(* IEC 61131-3 sources: SRCI/RobotLibrary/Library/POUs/General/MC_RobotTask (part 4) *)

         // timeout exceeded ?
         IF (CheckTimeout(_rTimer) = RobotLibraryConstants.OK)
         THEN
           ErrorID     := RobotLibraryErrorIdEnum.ERR_TIMEOUT_CMD;
           ErrorAddTxt := CONCAT(_stepName, DINT_TO_STRING(_rStep));
         END_IF
       END_IF

       // Wait Tooldata read
    2: IF (( NOT _readToolData.Busy  ) AND
           ( NOT _readToolData.Error ) AND
           (     _readToolData.Done  ))
       THEN
         // reset execution
        _readToolData.Execute := FALSE;
         // set available bit
        _toolData[_rSyncIdx].Available := TRUE;
         ToolData[_rSyncIdx].Available := TRUE;
         // Copy data
        _toolData[_rSyncIdx].Data := _readToolData.OutCmd.ToolData;

         // Check tool data is equal ?
         IF ( NOT IsToolDataEqual( Data1 := _toolData[_rSyncIdx].Data, Data2 := ToolData[_rSyncIdx].Data, IgnoreTimestamp := TRUE))
         THEN
           // Reset plc in sync flag
           AxesGroup.State.SyncStatePlc.InSync.Tool := FALSE;
           // Set data changed flag
           AxesGroup.State.DataChanged.Tool[_rSyncIdx] := TRUE;
           // inc count of unsynchronised plc tools
           AxesGroup.State.SyncStatePlc.UnSyncNo.Tool := AxesGroup.State.SyncStatePlc.UnSyncNo.Tool + 1;

           // Create log entry
           CreateLogMessagePara1 ( Timestamp   := SystemTime,
                                   MessageType := MessageType.CMD,
                                   Severity    := Severity.DEBUG,
                                   MessageCode := 0,
                                   MessageText := 'SyncToolData: Detected a difference in Tool[{1}] between PLC and RC',
                                   Para1       :=  DINT_TO_STRING(_rSyncIdx));

           // Check synchronisation is enabled ?
           IF ( NOT AxesGroup.State.DataEnableSync.EnableSyncTool ) AND (InfoID = RobotLibraryInfoIdEnum.NO_INFO )
           THEN
             InfoID := RobotLibraryInfoIdEnum.INFO_SYNC_TOOL_DATA_DISABLED;
  				 END_IF

           // Check user interaction needed ?
           IF ( AxesGroup.Parameter.PLC.Parameter.SyncUserInteraction.Tool ) AND ( WarningID = RobotLibraryWarningIdEnum.NO_WARNING )
           THEN
             WarningID := RobotLibraryWarningIdEnum.WARN_TOOL_NUMBER_SYNC_ERROR;
  				 END_IF
  			 END_IF

         // Check all tools read ?
         IF ( _rSyncIdx < AxesGroup.State.UnifiedToolIndex )
         THEN
           // set timeout
           SetTimeout(PT := _rTimeout, rTimer := _rTimer);
           // inc tool index
          _rSyncIdx := _rSyncIdx + 1;
           // dec step counter
          _rStep := _rStep - 1;
         ELSE
           // set timeout
           SetTimeout(PT := _rTimeout, rTimer := _rTimer);
           // inc step counter
          _rStep := _rStep + 1;
         END_IF
       ELSE
         // check error ?
         IF (_readToolData.Error)
         THEN
           // Set warning
           WarningID := RobotLibraryWarningIdEnum.WARN_TOOL_SYNC_FAILED_BY_ERROR_OF_READ_OR_WRITE_CMD;
           // reset available bit
           ToolData[_rSyncIdx].Available := FALSE;
          _toolData[_rSyncIdx].Available := FALSE;
         END_IF

         // timeout exceeded ?
         IF (CheckTimeout(_rTimer) = RobotLibraryConstants.OK)
         THEN
           ErrorID     := RobotLibraryErrorIdEnum.ERR_TIMEOUT_CMD;
           ErrorAddTxt := CONCAT(_stepName, DINT_TO_STRING(_rStep));
         END_IF
       END_IF

       // Check synchronisation state ?
    3: IF (( AxesGroup.State.SyncStatePlc.UnSyncNo.Tool                                            = 0                           ) OR
           ( AxesGroup.Parameter.Plc.Parameter.SynchronizationModes.Tool[SyncTime.DURING_START_UP] = SyncMode.NO_SYNCHRONIZATION ))
       THEN
         // Update bit for data in sync
         AxesGroup.State.SyncStatePlc.InSync.Tool := (AxesGroup.State.SyncStatePlc.UnSyncNo.Tool = 0);
         // set timeout
         SetTimeout(PT := _rTimeout, rTimer := _rTimer);
         // inc step counter
        _rStep := 10; // -> jump to after startup

         // Create log entry
         CreateLogMessagePara1 ( Timestamp   := SystemTime,
                                 MessageType := MessageType.CMD,
                                 Severity    := Severity.DEBUG,
                                 MessageCode := 0,
                                 MessageText := 'SyncToolData: Synchronization Startup Phase done',
                                 Para1       :=  '' );
       ELSE
         // Check user interaction needed ?
         IF ( NOT AxesGroup.Parameter.PLC.Parameter.SyncUserInteraction.Tool )
         THEN
           CASE AxesGroup.Parameter.Plc.Parameter.SynchronizationModes.Tool[SyncTime.DURING_START_UP] OF

             SyncMode.SERVER_TO_CLIENT :

               // Overwrite PLC data with RC data
               ToolData := _toolData;
               // Reset data changed flags
               AxesGroup.State.DataChanged.Tool := _dataChangedNone.Tool;
               // Reset Synchronizing flag
               AxesGroup.State.Synchronizing.Tool := FALSE;
               // Set plc in sync flag
               AxesGroup.State.SyncStatePlc.InSync.Tool := TRUE;
               // Reset count of unsynchronised plc tools
               AxesGroup.State.SyncStatePlc.UnSyncNo.Tool := 0;
               // set timeout
               SetTimeout(PT := _rTimeout, rTimer := _rTimer);
               // inc step counter
              _rStep := 10; // -> jump to after startup

              // Create log entry
              CreateLogMessagePara3 ( Timestamp   := SystemTime,
                                      MessageType := MessageType.CMD,
                                      Severity    := Severity.DEBUG,
                                      MessageCode := 0,
                                      MessageText := 'SyncToolData: Synchronization of Tools triggered by StartUp-Compare, SyncMode = {2}, SyncTime = {3}, SyncDirection = RC -> PLC',
                                      Para1       :=  DINT_TO_STRING(_rSyncIdx),
                                      Para2       :=  SYNC_MODE_TO_STRING(AxesGroup.Parameter.Plc.Parameter.SynchronizationModes.Tool[SyncTime.DURING_START_UP]),
                                      Para3       :=  SYNC_TIME_TO_STRING(SyncTime.DURING_START_UP));
              // Create log entry
              CreateLogMessagePara1 ( Timestamp   := SystemTime,
                                      MessageType := MessageType.CMD,
                                      Severity    := Severity.DEBUG,
                                      MessageCode := 0,
                                      MessageText := 'SyncToolData: Applied the initial read tool data from RC',
                                      Para1       :=  '' );

  				   SyncMode.CLIENT_TO_SERVER : ;

               // Check conflicts to solve ?
               FOR _rSyncIdx := 0 TO AxesGroup.State.UnifiedToolIndex
               DO
                 IF ( AxesGroup.State.DataChanged.Tool[_rSyncIdx] )
                 THEN
                  _found := TRUE;
                   EXIT;
  		  			   END_IF
               END_FOR

               IF ( _found )
               THEN
                 // Reset plc in sync flag
                 AxesGroup.State.SyncStatePlc.InSync.Tool := FALSE;
                 // Set Synchronizing flag
                 AxesGroup.State.Synchronizing.Tool := TRUE;
                 // set timeout
                 SetTimeout(PT := _rTimeout, rTimer := _rTimer);
                 // inc step counter
                _rStep := _rStep +1; // -> write PLC data to RC
                 // Create log entry
                 CreateLogMessagePara3 ( Timestamp   := SystemTime,
                                         MessageType := MessageType.CMD,
                                         Severity    := Severity.DEBUG,
                                         MessageCode := 0,
                                         MessageText := 'SyncToolData: Synchronization of Tool[{1}] triggered by StartUp-Compare, SyncMode = {2}, SyncTime = {3}, SyncDirection = PLC -> RC',
                                         Para1       :=  DINT_TO_STRING(_rSyncIdx),
                                         Para2       :=  SYNC_MODE_TO_STRING(AxesGroup.Parameter.Plc.Parameter.SynchronizationModes.Tool[SyncTime.DURING_START_UP]),
                                         Para3       :=  SYNC_TIME_TO_STRING(SyncTime.DURING_START_UP));
               ELSE
                 // Reset data changed flags
                 AxesGroup.State.DataChanged.Tool := _dataChangedNone.Tool;
                 // Reset Synchronizing flag
                 AxesGroup.State.Synchronizing.Tool := FALSE;
                 // Set plc in sync flag
                 AxesGroup.State.SyncStatePlc.InSync.Tool := TRUE;
                 // Reset count of unsynchronised tools
                 AxesGroup.State.SyncStatePlc.UnSyncNo.Tool := 0;
                 // set timeout
                 SetTimeout(PT := _rTimeout, rTimer := _rTimer);
                 // inc step counter
                _rStep := 10; // -> jump to after startup
  				     END_IF
           ELSE
             // invalid sync mode for startup
             ErrorID := RobotLibraryErrorIdEnum.ERR_SYNC_MODE_INVALID;
   	       END_CASE
         END_IF
       END_IF

       // Start write tool data
    4: IF (( NOT _writeToolData.Busy  ) AND
           ( NOT _writeToolData.Error ))
       THEN
         // set command parameter
        _writeToolData.ParCmd.ToolNo   := _rSyncIdx;
        _writeToolData.ParCmd.ToolData :=  ToolData[_rSyncIdx].Data;
         // execute command
        _writeToolData.Execute := TRUE;
         // set timeout
         SetTimeout(PT := _rTimeout, rTimer := _rTimer);
         // inc step counter
        _rStep := _rStep + 1;
       ELSE
         // check error ?
         IF (_writeToolData.Error)
         THEN
           ErrorID     := _writeToolData.ErrorID;
           ErrorAddTxt := _writeToolData.ErrorAddTxt;;
         END_IF

         // timeout exceeded ?
         IF (CheckTimeout(_rTimer) = RobotLibraryConstants.OK)
         THEN
           ErrorID     := RobotLibraryErrorIdEnum.ERR_TIMEOUT_CMD;
           ErrorAddTxt := CONCAT(_stepName, DINT_TO_STRING(_rStep));
         END_IF
       END_IF

       // Wait tool data written ?
    5: IF (( NOT _writeToolData.Busy  ) AND
           ( NOT _writeToolData.Error ) AND
           (     _writeToolData.Done  ))
       THEN
         // execute command
        _writeToolData.Execute := FALSE;
         // apply tool data to internal tool data
        _toolData[_rSyncIdx] := ToolData[_rSyncIdx];
         // reset data changed bit
         AxesGroup.State.DataChanged.Tool[_rSyncIdx] := FALSE;
         // dec count of unsynchronised tools
         AxesGroup.State.SyncStatePlc.UnSyncNo.Tool := AxesGroup.State.SyncStatePlc.UnSyncNo.Tool - 1;
         // set timeout
         SetTimeout(PT := _rTimeout, rTimer := _rTimer);
         // dec step counter
        _rStep := _rStep - 2;
       ELSE
         // check error ?
         IF (_writeToolData.Error)
         THEN
           WarningID := RobotLibraryWarningIdEnum.WARN_TOOL_SYNC_FAILED_BY_ERROR_OF_READ_OR_WRITE_CMD;
         END_IF

         // timeout exceeded ?
         IF (CheckTimeout(_rTimer) = RobotLibraryConstants.OK)
         THEN
           ErrorID     := RobotLibraryErrorIdEnum.ERR_TIMEOUT_CMD;
           ErrorAddTxt := CONCAT(_stepName, DINT_TO_STRING(_rStep));
         END_IF
       END_IF

    // --------------------------------------------
    // SyncMode after startup :
    // --------------------------------------------

    10 :// check synchronisation active ?
         IF ( AxesGroup.Parameter.Plc.Parameter.SynchronizationModes.Tool[SyncTime.AFTER_START_UP] = SyncMode.NO_SYNCHRONIZATION)
         THEN
           RETURN;
         END_IF

         // reset count of unsynchronised tools
         AxesGroup.State.SyncStatePlc.UnSyncNo.Tool := 0;

         // Check all tool datas
         FOR _rSyncIdx := 0 TO AxesGroup.State.UnifiedToolIndex
         DO
           // compare tool data
           AxesGroup.State.DataChanged.Tool[_rSyncIdx] := NOT IsToolDataEqual( Data1 := ToolData[_rSyncIdx].Data, Data2 := _toolData[_rSyncIdx].Data, IgnoreTimestamp := FALSE);

           // Check Tool data changed ?
           IF (AxesGroup.State.DataChanged.Tool[_rSyncIdx])
           THEN
             // inc count of unsynchronised plc tools
             AxesGroup.State.SyncStatePlc.UnSyncNo.Tool := AxesGroup.State.SyncStatePlc.UnSyncNo.Tool + 1;
             // Create log entry
             CreateLogMessagePara2 ( Timestamp   := SystemTime,
                                     MessageType := MessageType.CMD,
                                     Severity    := Severity.DEBUG,
                                     MessageCode := 0,
                                     MessageText := 'SyncToolData: Detected a local change of Tool[{1}] on PLC, SyncTime = {2}',
                                     Para1       :=  DINT_TO_STRING(_rSyncIdx),
                                     Para2       :=  SYNC_TIME_TO_STRING(SyncTime.AFTER_START_UP));
  				 END_IF

           // Update plc in sync flag
           AxesGroup.State.SyncStatePlc.InSync.Tool := (AxesGroup.State.SyncStatePlc.UnSyncNo.Tool = 0);
  	     END_FOR

         // Check synchronization is needed ?
         IF ( NOT AxesGroup.State.SyncStatePlc.InSync.Tool ) XOR
            ( NOT AxesGroup.State.SyncStateRc .InSync.Tool )
         THEN
           CASE AxesGroup.Parameter.Plc.Parameter.SynchronizationModes.Tool[SyncTime.AFTER_START_UP]
           OF
             // NO_SYNCHRONIZATION
             SyncMode.NO_SYNCHRONIZATION : ; // no further action

             // CLIENT_TO_SERVER
             SyncMode.CLIENT_TO_SERVER :
               // set timeout
               SetTimeout(PT := _rTimeout, rTimer := _rTimer);
               // inc step counter
              _rStep := 11;

             // SERVER_TO_CLIENT
             SyncMode.SERVER_TO_CLIENT :
               // set timeout
               SetTimeout(PT := _rTimeout, rTimer := _rTimer);
               // inc step counter
              _rStep := 12;

             // AUTOMATIC
             SyncMode.AUTOMATIC :
               // set timeout
               SetTimeout(PT := _rTimeout, rTimer := _rTimer);
               // inc step counter
              _rStep := 13;
           END_CASE
         ELSE
           // datas changeḍ on both sides ? -> Warning
           IF (( NOT AxesGroup.State.SyncStatePlc.InSync.Tool ) AND
               ( NOT AxesGroup.State.SyncStateRc .InSync.Tool ))
           THEN
             WarningID := RobotLibraryWarningIdEnum.WARN_TOOL_SYNC_BOTH_SIDES_CHANGED;
           END_IF
         END_IF

    // ------------------------------------------
    // SyncMode : CLIENT_TO_SERVER
    // ------------------------------------------
    11 : // Conflict triggerd by PLC ?
         IF ( NOT AxesGroup.State.SyncStatePlc.InSync.Tool )
         THEN
           // search for changed index
           FOR _rSyncIdx := 0 TO AxesGroup.State.UnifiedToolIndex
           DO
             IF ( AxesGroup.State.DataChanged.Tool[_rSyncIdx] )
             THEN
               // set timeout
               SetTimeout(PT := _rTimeout, rTimer := _rTimer);
               // inc step counter
              _rStep := 30; // -> write PLC data to RC
               EXIT;
  					 END_IF
           END_FOR

           // Create log entry
           CreateLogMessagePara3 ( Timestamp   := SystemTime,
                                   MessageType := MessageType.CMD,
                                   Severity    := Severity.DEBUG,
                                   MessageCode := 0,
                                   MessageText := 'SyncToolData: Synchronization of Tool[{1}] triggered by PLC, SyncMode = {2}, SyncTime = {3}, SyncDirection = PLC -> RC',
                                   Para1       :=  DINT_TO_STRING(_rSyncIdx),
                                   Para2       :=  SYNC_MODE_TO_STRING(AxesGroup.Parameter.Plc.Parameter.SynchronizationModes.Tool[SyncTime.AFTER_START_UP]),
                                   Para3       :=  SYNC_TIME_TO_STRING(SyncTime.AFTER_START_UP));
                                   RETURN;
         END_IF

         // Conflict triggered by RC ?
         IF ( NOT AxesGroup.State.SyncStateRc.InSync.Tool )
         THEN
           // get changed index
          _rSyncIdx :=  LIMIT(0, AxesGroup.State.SyncStateRc.UnSyncNo.Tool, AxesGroup.State.UnifiedToolIndex);
           // set timeout
           SetTimeout(PT := _rTimeout, rTimer := _rTimer);
           // inc step counter
          _rStep := 30; // -> write PLC data to RC

           // Create log entry
           CreateLogMessagePara3 ( Timestamp   := SystemTime,
                                   MessageType := MessageType.CMD,
                                   Severity    := Severity.DEBUG,
                                   MessageCode := 0,
                                   MessageText := 'SyncToolData: Synchronization of Tool[{1}] triggered by RC, SyncMode = {2}, SyncTime = {3}, SyncDirection = PLC -> RC',
                                   Para1       :=  DINT_TO_STRING(_rSyncIdx),
                                   Para2       :=  SYNC_MODE_TO_STRING(AxesGroup.Parameter.Plc.Parameter.SynchronizationModes.Tool[SyncTime.AFTER_START_UP]),
                                   Para3       :=  SYNC_TIME_TO_STRING(SyncTime.AFTER_START_UP));
                                   RETURN;
  			 END_IF

         // set timeout
         SetTimeout(PT := _rTimeout, rTimer := _rTimer);
         // jump back
        _rStep := 10;

    // ------------------------------------------
    // SyncMode : SERVER_TO_CLIENT
    // ------------------------------------------
    12 : // Conflict triggerd by PLC ?
         IF ( NOT AxesGroup.State.SyncStatePlc.InSync.Tool )
         THEN
           // search for changed index
           FOR _rSyncIdx := 0 TO AxesGroup.State.UnifiedToolIndex
           DO
             IF ( AxesGroup.State.DataChanged.Tool[_rSyncIdx] )
             THEN
               // set timeout
               SetTimeout(PT := _rTimeout, rTimer := _rTimer);
               // inc step counter
              _rStep := 20; // -> read RC data and write it to PLC
               EXIT;
  					 END_IF
           END_FOR

           // Create log entry
           CreateLogMessagePara3 ( Timestamp   := SystemTime,
                                   MessageType := MessageType.CMD,
                                   Severity    := Severity.DEBUG,
                                   MessageCode := 0,
                                   MessageText := 'SyncToolData: Synchronization of Tool[{1}] triggered by PLC, SyncMode = {2}, SyncTime = {3}, SyncDirection = RC -> PLC',
                                   Para1       :=  DINT_TO_STRING(_rSyncIdx),
                                   Para2       :=  SYNC_MODE_TO_STRING(AxesGroup.Parameter.Plc.Parameter.SynchronizationModes.Tool[SyncTime.AFTER_START_UP]),
                                   Para3       :=  SYNC_TIME_TO_STRING(SyncTime.AFTER_START_UP));
                                   RETURN;
         END_IF

         // Conflict triggered by RC ?
         IF ( NOT AxesGroup.State.SyncStateRc.InSync.Tool )
         THEN
           // get changed index
          _rSyncIdx := LIMIT(0, AxesGroup.State.SyncStateRc.UnSyncNo.Tool, AxesGroup.State.UnifiedToolIndex);
           // set timeout
           SetTimeout(PT := _rTimeout, rTimer := _rTimer);
           // inc step counter
          _rStep := 20; // -> read RC data and write it to PLC

           // Create log entry
           CreateLogMessagePara3 ( Timestamp   := SystemTime,
                                   MessageType := MessageType.CMD,
                                   Severity    := Severity.DEBUG,
                                   MessageCode := 0,
                                   MessageText := 'SyncToolData: Synchronization of Tool[{1}] triggered by RC, SyncMode = {2}, SyncTime = {3}, SyncDirection = RC -> PLC',
                                   Para1       :=  DINT_TO_STRING(_rSyncIdx),
                                   Para2       :=  SYNC_MODE_TO_STRING(AxesGroup.Parameter.Plc.Parameter.SynchronizationModes.Tool[SyncTime.AFTER_START_UP]),
                                   Para3       :=  SYNC_TIME_TO_STRING(SyncTime.AFTER_START_UP));
                                   RETURN;
  			 END_IF

         // set timeout
         SetTimeout(PT := _rTimeout, rTimer := _rTimer);
         // jump back
        _rStep := 10;

    // ------------------------------------------
    // SyncMode : AUTOMATIC
    // ------------------------------------------
    13 : // Conflict triggerd by PLC ?
         IF ( NOT AxesGroup.State.SyncStatePlc.InSync.Tool )
         THEN
           // search for changed index
           FOR _rSyncIdx := 0 TO AxesGroup.State.UnifiedToolIndex
           DO
             IF ( AxesGroup.State.DataChanged.Tool[_rSyncIdx] )
             THEN
               // set timeout
               SetTimeout(PT := _rTimeout, rTimer := _rTimer);
               // inc step counter
              _rStep := 30; // -> write PLC data to RC
               EXIT;
  					 END_IF
           END_FOR

           // Create log entry
           CreateLogMessagePara3 ( Timestamp   := SystemTime,
                                   MessageType := MessageType.CMD,
                                   Severity    := Severity.DEBUG,
                                   MessageCode := 0,
                                   MessageText := 'SyncToolData: Synchronization of Tool[{1}] triggered by PLC, SyncMode = {2}, SyncTime = {3}, SyncDirection = PLC -> RC',
                                   Para1       :=  DINT_TO_STRING(_rSyncIdx),
                                   Para2       :=  SYNC_MODE_TO_STRING(AxesGroup.Parameter.Plc.Parameter.SynchronizationModes.Tool[SyncTime.AFTER_START_UP]),
                                   Para3       :=  SYNC_TIME_TO_STRING(SyncTime.AFTER_START_UP));
                                   RETURN;
         END_IF

         // Conflict triggered by RC ?
         IF ( NOT AxesGroup.State.SyncStateRc.InSync.Tool )
         THEN
           // get changed index
          _rSyncIdx := LIMIT(0, AxesGroup.State.SyncStateRc.UnSyncNo.Tool, AxesGroup.State.UnifiedToolIndex);
           // set timeout
           SetTimeout(PT := _rTimeout, rTimer := _rTimer);
           // inc step counter
          _rStep := 20; // -> read RC data an write it to PLC

           // Create log entry
           CreateLogMessagePara3 ( Timestamp   := SystemTime,
                                   MessageType := MessageType.CMD,
                                   Severity    := Severity.DEBUG,
                                   MessageCode := 0,
                                   MessageText := 'SyncToolData: Synchronization of Tool[{1}] triggered by RC, SyncMode = {2}, SyncTime = {3}, SyncDirection = RC -> PLC',
                                   Para1       :=  DINT_TO_STRING(_rSyncIdx),
                                   Para2       :=  SYNC_MODE_TO_STRING(AxesGroup.Parameter.Plc.Parameter.SynchronizationModes.Tool[SyncTime.AFTER_START_UP]),
                                   Para3       :=  SYNC_TIME_TO_STRING(SyncTime.AFTER_START_UP));
                                   RETURN;
  			 END_IF

         // set timeout
         SetTimeout(PT := _rTimeout, rTimer := _rTimer);
         // jump back
        //_rStep := 10;

    // ------------------------------------------
    // Read Data from RC and write it to PLC
    // ------------------------------------------
    20 : IF (( NOT _readToolData.Busy  ) AND
             ( NOT _readToolData.Error ))
         THEN
           // set command parameter
          _readToolData.ParCmd.ToolNo := _rSyncIdx;
           // execute command
          _readToolData.Execute := TRUE;
           // set timeout
           SetTimeout(PT := _rTimeout, rTimer := _rTimer);
           // inc step counter
          _rStep := _rStep + 1;
         ELSE
           // check error ?
           IF (_readToolData.Error)
           THEN
             ErrorID     := _readToolData.ErrorID;
             ErrorAddTxt := _readToolData.ErrorAddTxt;
           END_IF

           // timeout exceeded ?
           IF (CheckTimeout(_rTimer) = RobotLibraryConstants.OK)
           THEN
             ErrorID     := RobotLibraryErrorIdEnum.ERR_TIMEOUT_CMD;
             ErrorAddTxt := CONCAT(_stepName, DINT_TO_STRING(_rStep));
           END_IF
         END_IF

    21 : IF (( NOT _readToolData.Busy  ) AND
             ( NOT _readToolData.Error ) AND
             (     _readToolData.Done  ))
         THEN
           // reset execution
          _readToolData.Execute := FALSE;
           // update internal tool data
           ToolData[_rSyncIdx].Data := _readToolData.OutCmd.ToolData;
          _toolData[_rSyncIdx].Data := _readToolData.OutCmd.ToolData;
           // set available bit
           ToolData[_rSyncIdx].Available := TRUE;
          _toolData[_rSyncIdx].Available := TRUE;
           // set timeout
           SetTimeout(PT := _rTimeout, rTimer := _rTimer);
           // inc step counter
          _rStep := 10; // -> jump to after startup
         ELSE
           // check error ?
           IF (_readToolData.Error)
           THEN
             ErrorID     := _readToolData.ErrorID;
             ErrorAddTxt := _readToolData.ErrorAddTxt;
             // reset available bit
             ToolData[_rSyncIdx].Available := FALSE;
            _toolData[_rSyncIdx].Available := FALSE;
           END_IF

           // timeout exceeded ?
           IF (CheckTimeout(_rTimer) = RobotLibraryConstants.OK)
           THEN
             ErrorID     := RobotLibraryErrorIdEnum.ERR_TIMEOUT_CMD;
             ErrorAddTxt := CONCAT(_stepName, DINT_TO_STRING(_rStep));
           END_IF
         END_IF

    // ------------------------------------------
    // Write data from PLC to RC
    // ------------------------------------------
    30 : IF (( NOT _writeToolData.Busy  ) AND
             ( NOT _writeToolData.Error ))
         THEN
           // set command parameter
          _writeToolData.ParCmd.ToolNo   := _rSyncIdx;
          _writeToolData.ParCmd.ToolData :=  ToolData[_rSyncIdx].Data;
           // execute command
          _writeToolData.Execute := TRUE;
           // set timeout
           SetTimeout(PT := _rTimeout, rTimer := _rTimer);
           // inc step counter
          _rStep := _rStep + 1;
         ELSE
           // check error ?
           IF (_writeToolData.Error)
           THEN
             ErrorID     := _writeToolData.ErrorID;
             ErrorAddTxt := _writeToolData.ErrorAddTxt;;
           END_IF

           // timeout exceeded ?
           IF (CheckTimeout(_rTimer) = RobotLibraryConstants.OK)
           THEN
             ErrorID     := RobotLibraryErrorIdEnum.ERR_TIMEOUT_CMD;
             ErrorAddTxt := CONCAT(_stepName, DINT_TO_STRING(_rStep));
           END_IF
         END_IF

    31 : IF (( NOT _writeToolData.Busy  ) AND
             ( NOT _writeToolData.Error ) AND
             (     _writeToolData.Done  ))
         THEN
           // execute command
          _writeToolData.Execute := FALSE;
           // update internal tool data
          _toolData[_rSyncIdx] := ToolData[_rSyncIdx];
           // set available bit
           ToolData[_rSyncIdx].Available := TRUE;
          _toolData[_rSyncIdx].Available := TRUE;
           // set timeout
           SetTimeout(PT := _rTimeout, rTimer := _rTimer);
           // inc step counter
          _rStep := 10; // -> jump to after startup;
         ELSE
           // check error ?
           IF (_writeToolData.Error)
           THEN
             WarningID := RobotLibraryWarningIdEnum.WARN_TOOL_SYNC_FAILED_BY_ERROR_OF_READ_OR_WRITE_CMD;
             // reset available bit
             ToolData[_rSyncIdx].Available := FALSE;
            _toolData[_rSyncIdx].Available := FALSE;
           END_IF

           // timeout exceeded ?
           IF (CheckTimeout(_rTimer) = RobotLibraryConstants.OK)
           THEN
             ErrorID     := RobotLibraryErrorIdEnum.ERR_TIMEOUT_CMD;
             ErrorAddTxt := CONCAT(_stepName, DINT_TO_STRING(_rStep));
           END_IF
         END_IF

  ELSE
    // invalid step
    ErrorID     := RobotLibraryErrorIdEnum.ERR_INVALID_STEP;
    ErrorAddTxt := CONCAT(_stepName , DINT_TO_STRING(_stepCmd));
  END_CASE

END_METHOD

METHOD PRIVATE HandleSyncWorkArea
VAR_IN_OUT
   /// Robot assignment of function
  AxesGroup : AxesGroup;
  /// Work areas stored on PLC. For more information refer to 5.5.8
  WorkAreas : ARRAY[0..RobotLibraryParameter.WORK_AREAS_MAX -1] OF RobotWorkArea;
END_VAR

VAR
  /// Internal step counter name
 _stepName        : STRING;
  /// Internal reference to step counter
 _rStep           : REFERENCE TO DINT;
  /// Internal reference to timer
 _rTimer          : REFERENCE TO TON;
  /// Internal reference to timeout
 _rTimeout        : REFERENCE TO TIME;
  /// Internal reference to synchroniztion index
 _rSyncIdx        : REFERENCE TO USINT;
  /// internal bit for condition found
 _found           : BOOL;
  /// empty data set to reset all DataChanged bits
 _dataChangedNone : AxesGroupStateDataChanged;
END_VAR

  // Set internal references
  _stepName      :=   '_stepSyncWorkArea = ';
  _rStep       REF=    _stepSyncWorkArea;
  _rTimer      REF=   _timerSyncWorkArea;
  _rTimeout    REF= _timeoutSyncWorkArea;
  _rSyncIdx    REF=     _syncIdxWorkArea;

  CASE _rStep
  OF
    0: // Check initialisation configured ?
       IF (( _parCfg.PLC.Parameter.SynchronizationModes.WorkAreas[SyncTime.DURING_START_UP] = SyncMode.NO_SYNCHRONIZATION ) AND
           ( _parCfg.PLC.Parameter.SynchronizationModes.WorkAreas[SyncTime. AFTER_START_UP] = SyncMode.NO_SYNCHRONIZATION ))
       THEN
         RETURN;
       END_IF

       // wait for initialisation done
       IF  ((     AxesGroup.State.RobotData.RCSupportedFunctions. ReadWorkArea ) AND
            (     AxesGroup.State.RobotData.RCSupportedFunctions.WriteWorkArea ) AND
            (     AxesGroup.State.Initialized                                  ) AND
            ( NOT Error                                                        ))
       THEN
         // Check PLC WorkAreas < RC WorkAreas and SyncWorkArea enabled ?
         IF (( AxesGroup.State.DataEnableSync.EnableSyncWorkArea      = TRUE                                    )  AND
             ( AxesGroup.Parameter.Rob.Parameter.HighestWorkAreaIndex > RobotLibraryParameter.WORK_AREAS_MAX -1 ))
         THEN
           WarningID := RobotLibraryWarningIdEnum.WARN_WORK_AREA_ARRAY_TOO_SHORT;
         END_IF

         // Create log entry
         CreateLogMessagePara1 ( Timestamp   := SystemTime,
                                 MessageType := MessageType.CMD,
                                 Severity    := Severity.DEBUG,
                                 MessageCode := 0,
                                 MessageText := 'SyncWorkArea: Start initial reading of WorkArea from RC',
                                 Para1       :=  '');

         // init WorkArea number
        _rSyncIdx := 0;
         // init count of unsynchronized elements
         AxesGroup.State.SyncStatePlc.UnSyncNo.WorkArea := 0;
         // set timeout
         SetTimeout(PT := _rTimeout, rTimer := _rTimer);
         // inc step counter
        _rStep := _rStep + 1;
       END_IF

       // Start read WorkArea
    1: IF (( NOT _readWorkArea.Busy  ) AND
           ( NOT _readWorkArea.Error ))
       THEN
         // set command parameter
        _readWorkArea.ParCmd.WorkAreaNo := _rSyncIdx;
         // execute command
        _readWorkArea.Execute := TRUE;
         // set timeout
         SetTimeout(PT := _rTimeout, rTimer := _rTimer);
         // inc step counter
        _rStep := _rStep + 1;
       ELSE
         // check error ?
         IF ( _readWorkArea.Error ) AND ( WarningID = RobotLibraryWarningIdEnum.NO_WARNING )
         THEN
           WarningID := RobotLibraryWarningIdEnum.WARN_WORK_AREA_SYNC_FAILED_BY_ERROR_OF_READ_OR_WRITE_CMD;
         END_IF

         // timeout exceeded ?
         IF (CheckTimeout(_rTimer) = RobotLibraryConstants.OK)
         THEN
           ErrorID     := RobotLibraryErrorIdEnum.ERR_TIMEOUT_CMD;
           ErrorAddTxt := CONCAT(_stepName, DINT_TO_STRING(_rStep));
         END_IF
       END_IF

       // Wait WorkArea read
    2: IF (( NOT _readWorkArea.Busy  ) AND
           ( NOT _readWorkArea.Error ) AND
           (     _readWorkArea.Done  ))
       THEN
         // reset execution
        _readWorkArea.Execute := FALSE;
         // set available bit
        _workAreas[_rSyncIdx].Available := TRUE;
         WorkAreas[_rSyncIdx].Available := TRUE;
         // Copy data
        _workAreas[_rSyncIdx].Data := _readWorkArea.OutCmd.WorkAreaData;

         // Check WorkArea data is equal ?
         IF ( NOT IsWorkAreaEqual( Data1 := _workAreas[_rSyncIdx].Data, Data2 := WorkAreas[_rSyncIdx].Data, IgnoreTimestamp := TRUE))
         THEN
           // Reset plc in sync flag
           AxesGroup.State.SyncStatePlc.InSync.WorkArea := FALSE;
           // Set data changed flag
           AxesGroup.State.DataChanged.WorkArea[_rSyncIdx] := TRUE;
           // inc count of unsynchronised plc WorkAreas
           AxesGroup.State.SyncStatePlc.UnSyncNo.WorkArea := AxesGroup.State.SyncStatePlc.UnSyncNo.WorkArea + 1;

           // Create log entry
           CreateLogMessagePara1 ( Timestamp   := SystemTime,
                                   MessageType := MessageType.CMD,
                                   Severity    := Severity.DEBUG,
                                   MessageCode := 0,
                                   MessageText := 'SyncWorkArea: Detected a difference in WorkArea[{1}] between PLC and RC',
                                   Para1       :=  DINT_TO_STRING(_rSyncIdx));

           // Check synchronisation is enabled ?
           IF ( NOT AxesGroup.State.DataEnableSync.EnableSyncWorkArea ) AND (InfoID = RobotLibraryInfoIdEnum.NO_INFO )
           THEN
             InfoID := RobotLibraryInfoIdEnum.INFO_SYNC_WORK_AREA_DISABLED;
  				 END_IF

           // Check user interaction needed ?
           IF ( AxesGroup.Parameter.PLC.Parameter.SyncUserInteraction.WorkAreas ) AND ( WarningID = RobotLibraryWarningIdEnum.NO_WARNING )
           THEN
             WarningID := RobotLibraryWarningIdEnum.WARN_WORK_AREA_NUMBER_SYNC_ERROR;
  				 END_IF
  			 END_IF

         // Check all WorkAreas read ?
         IF ( _rSyncIdx < AxesGroup.State.UnifiedWorkAreaIndex )
         THEN
           // set timeout
           SetTimeout(PT := _rTimeout, rTimer := _rTimer);
           // inc WorkArea index
          _rSyncIdx := _rSyncIdx + 1;
           // dec step counter
          _rStep := _rStep - 1;
         ELSE
           // set timeout
           SetTimeout(PT := _rTimeout, rTimer := _rTimer);
           // inc step counter
          _rStep := _rStep + 1;
         END_IF
       ELSE
         // check error ?
         IF (_readWorkArea.Error)
         THEN
           // Set warning
           WarningID := RobotLibraryWarningIdEnum.WARN_WORK_AREA_SYNC_FAILED_BY_ERROR_OF_READ_OR_WRITE_CMD;
           // reset available bit
           WorkAreas[_rSyncIdx].Available := FALSE;
          _workAreas[_rSyncIdx].Available := FALSE;
         END_IF

         // timeout exceeded ?
         IF (CheckTimeout(_rTimer) = RobotLibraryConstants.OK)
         THEN
           ErrorID     := RobotLibraryErrorIdEnum.ERR_TIMEOUT_CMD;
           ErrorAddTxt := CONCAT(_stepName, DINT_TO_STRING(_rStep));
         END_IF
       END_IF

       // Check synchronisation state ?
    3: IF (( AxesGroup.State.SyncStatePlc.UnSyncNo.WorkArea                                             = 0                           ) OR
           ( AxesGroup.Parameter.Plc.Parameter.SynchronizationModes.WorkAreas[SyncTime.DURING_START_UP] = SyncMode.NO_SYNCHRONIZATION ))
       THEN
         // Update bit for data in sync
         AxesGroup.State.SyncStatePlc.InSync.WorkArea := (AxesGroup.State.SyncStatePlc.UnSyncNo.WorkArea = 0);
         // set timeout
         SetTimeout(PT := _rTimeout, rTimer := _rTimer);
         // inc step counter
        _rStep := 10; // -> jump to after startup

         // Create log entry
         CreateLogMessagePara1 ( Timestamp   := SystemTime,
                                 MessageType := MessageType.CMD,
                                 Severity    := Severity.DEBUG,
                                 MessageCode := 0,
                                 MessageText := 'SyncWorkArea: Synchronization Startup Phase done',
                                 Para1       :=  '' );
       ELSE
         // Check user interaction needed ?
         IF ( NOT AxesGroup.Parameter.PLC.Parameter.SyncUserInteraction.WorkAreas )
         THEN
           CASE AxesGroup.Parameter.Plc.Parameter.SynchronizationModes.WorkAreas[SyncTime.DURING_START_UP] OF

             SyncMode.SERVER_TO_CLIENT :

               // Overwrite PLC data with RC data
               WorkAreas := _workAreas;
               // Reset data changed flags
               AxesGroup.State.DataChanged.WorkArea := _dataChangedNone.WorkArea;
               // Reset Synchronizing flag
               AxesGroup.State.Synchronizing.WorkAreas := FALSE;
               // Set plc in sync flag
               AxesGroup.State.SyncStatePlc.InSync.WorkArea := TRUE;
               // Reset count of unsynchronised plc WorkAreas
               AxesGroup.State.SyncStatePlc.UnSyncNo.WorkArea := 0;
               // set timeout
               SetTimeout(PT := _rTimeout, rTimer := _rTimer);
               // inc step counter
              _rStep := 10; // -> jump to after startup

              // Create log entry
              CreateLogMessagePara3 ( Timestamp   := SystemTime,
                                      MessageType := MessageType.CMD,
                                      Severity    := Severity.DEBUG,
                                      MessageCode := 0,
                                      MessageText := 'SyncWorkArea: Synchronization of WorkAreas triggered by StartUp-Compare, SyncMode = {2}, SyncTime = {3}, SyncDirection = RC -> PLC',
                                      Para1       :=  DINT_TO_STRING(_rSyncIdx),
                                      Para2       :=  SYNC_MODE_TO_STRING(AxesGroup.Parameter.Plc.Parameter.SynchronizationModes.WorkAreas[SyncTime.DURING_START_UP]),
                                      Para3       :=  SYNC_TIME_TO_STRING(SyncTime.DURING_START_UP));
              // Create log entry
              CreateLogMessagePara1 ( Timestamp   := SystemTime,
                                      MessageType := MessageType.CMD,
                                      Severity    := Severity.DEBUG,
                                      MessageCode := 0,
                                      MessageText := 'SyncWorkArea: Applied the initial read WorkArea data from RC',
                                      Para1       :=  '' );

  				   SyncMode.CLIENT_TO_SERVER : ;

               // Check conflicts to solve ?
               FOR _rSyncIdx := 0 TO AxesGroup.State.UnifiedWorkAreaIndex
               DO
                 IF ( AxesGroup.State.DataChanged.WorkArea[_rSyncIdx] )
                 THEN
                  _found := TRUE;
                   EXIT;
  		  			   END_IF
               END_FOR

               IF ( _found )
               THEN
                 // Reset plc in sync flag
                 AxesGroup.State.SyncStatePlc.InSync.WorkArea := FALSE;
                 // Set Synchronizing flag
                 AxesGroup.State.Synchronizing.WorkAreas := TRUE;
                 // set timeout
                 SetTimeout(PT := _rTimeout, rTimer := _rTimer);
                 // inc step counter
                _rStep := _rStep +1; // -> write PLC data to RC
                 // Create log entry
                 CreateLogMessagePara3 ( Timestamp   := SystemTime,
                                         MessageType := MessageType.CMD,
                                         Severity    := Severity.DEBUG,
                                         MessageCode := 0,
                                         MessageText := 'SyncWorkArea: Synchronization of WorkArea[{1}] triggered by StartUp-Compare, SyncMode = {2}, SyncTime = {3}, SyncDirection = PLC -> RC',
                                         Para1       :=  DINT_TO_STRING(_rSyncIdx),
                                         Para2       :=  SYNC_MODE_TO_STRING(AxesGroup.Parameter.Plc.Parameter.SynchronizationModes.WorkAreas[SyncTime.DURING_START_UP]),
                                         Para3       :=  SYNC_TIME_TO_STRING(SyncTime.DURING_START_UP));
               ELSE
                 // Reset data changed flags
                 AxesGroup.State.DataChanged.WorkArea := _dataChangedNone.WorkArea;
                 // Reset Synchronizing flag
                 AxesGroup.State.Synchronizing.WorkAreas := FALSE;
                 // Set plc in sync flag
                 AxesGroup.State.SyncStatePlc.InSync.WorkArea := TRUE;
                 // Reset count of unsynchronised WorkAreas
                 AxesGroup.State.SyncStatePlc.UnSyncNo.WorkArea := 0;
                 // set timeout
                 SetTimeout(PT := _rTimeout, rTimer := _rTimer);
                 // inc step counter
                _rStep := 10; // -> jump to after startup
  				     END_IF
           ELSE
             // invalid sync mode for startup
             ErrorID := RobotLibraryErrorIdEnum.ERR_SYNC_MODE_INVALID;
   	       END_CASE
         END_IF
       END_IF

       // Start write WorkArea data
    4: IF (( NOT _writeWorkArea.Busy  ) AND
           ( NOT _writeWorkArea.Error ))
       THEN
         // set command parameter
        _writeWorkArea.ParCmd.WorkAreaNo   := _rSyncIdx;
        _writeWorkArea.ParCmd.WorkAreaData :=  WorkAreas[_rSyncIdx].Data;
         // execute command
        _writeWorkArea.Execute := TRUE;
         // set timeout
         SetTimeout(PT := _rTimeout, rTimer := _rTimer);
         // inc step counter
        _rStep := _rStep + 1;
       ELSE
         // check error ?
         IF (_writeWorkArea.Error)
         THEN
           ErrorID     := _writeWorkArea.ErrorID;
           ErrorAddTxt := _writeWorkArea.ErrorAddTxt;;
         END_IF

         // timeout exceeded ?
         IF (CheckTimeout(_rTimer) = RobotLibraryConstants.OK)
         THEN
           ErrorID     := RobotLibraryErrorIdEnum.ERR_TIMEOUT_CMD;
           ErrorAddTxt := CONCAT(_stepName, DINT_TO_STRING(_rStep));
         END_IF
       END_IF

       // Wait WorkArea data written ?
    5: IF (( NOT _writeWorkArea.Busy  ) AND
           ( NOT _writeWorkArea.Error ) AND
           (     _writeWorkArea.Done  ))
       THEN
         // execute command
        _writeWorkArea.Execute := FALSE;
         // apply WorkArea data to internal WorkArea data
        _workAreas[_rSyncIdx] := WorkAreas[_rSyncIdx];
         // reset data changed bit
         AxesGroup.State.DataChanged.WorkArea[_rSyncIdx] := FALSE;
         // dec count of unsynchronised WorkAreas
         AxesGroup.State.SyncStatePlc.UnSyncNo.WorkArea := AxesGroup.State.SyncStatePlc.UnSyncNo.WorkArea - 1;
         // set timeout
         SetTimeout(PT := _rTimeout, rTimer := _rTimer);
         // dec step counter
        _rStep := _rStep - 2;
       ELSE
         // check error ?
         IF (_writeWorkArea.Error)
         THEN
           WarningID := RobotLibraryWarningIdEnum.WARN_WORK_AREA_SYNC_FAILED_BY_ERROR_OF_READ_OR_WRITE_CMD;
         END_IF

         // timeout exceeded ?
         IF (CheckTimeout(_rTimer) = RobotLibraryConstants.OK)
         THEN
           ErrorID     := RobotLibraryErrorIdEnum.ERR_TIMEOUT_CMD;
           ErrorAddTxt := CONCAT(_stepName, DINT_TO_STRING(_rStep));
         END_IF
       END_IF

    // --------------------------------------------
    // SyncMode after startup :
    // --------------------------------------------

    10 : // check synchronisation active ?
         IF ( AxesGroup.Parameter.Plc.Parameter.SynchronizationModes.WorkAreas[SyncTime.AFTER_START_UP] = SyncMode.NO_SYNCHRONIZATION)
         THEN
           RETURN;
         END_IF

         // reset count of unsynchronised WorkAreas
         AxesGroup.State.SyncStatePlc.UnSyncNo.WorkArea := 0;

         // Check all WorkArea datas
         FOR _rSyncIdx := 0 TO AxesGroup.State.UnifiedWorkAreaIndex
         DO
           // compare WorkArea data
           AxesGroup.State.DataChanged.WorkArea[_rSyncIdx] := NOT IsWorkAreaEqual( Data1 := WorkAreas[_rSyncIdx].Data, Data2 := _workAreas[_rSyncIdx].Data, IgnoreTimestamp := FALSE);

           // Check WorkArea data changed ?
           IF (AxesGroup.State.DataChanged.WorkArea[_rSyncIdx])
           THEN
             // inc count of unsynchronised plc WorkAreas
             AxesGroup.State.SyncStatePlc.UnSyncNo.WorkArea := AxesGroup.State.SyncStatePlc.UnSyncNo.WorkArea + 1;
             // Create log entry
             CreateLogMessagePara2 ( Timestamp   := SystemTime,
                                     MessageType := MessageType.CMD,
                                     Severity    := Severity.DEBUG,
                                     MessageCode := 0,
                                     MessageText := 'SyncWorkArea: Detected a local change of WorkArea[{1}] on PLC, SyncTime = {2}',
                                     Para1       :=  DINT_TO_STRING(_rSyncIdx),
                                     Para2       :=  SYNC_TIME_TO_STRING(SyncTime.AFTER_START_UP));
  				 END_IF

           // Update plc in sync flag
           AxesGroup.State.SyncStatePlc.InSync.WorkArea := (AxesGroup.State.SyncStatePlc.UnSyncNo.WorkArea = 0);
  	     END_FOR

         // Check synchronization is needed ?
         IF ( NOT AxesGroup.State.SyncStatePlc.InSync.WorkArea ) XOR
            ( NOT AxesGroup.State.SyncStateRc .InSync.WorkArea )
         THEN
           CASE AxesGroup.Parameter.Plc.Parameter.SynchronizationModes.WorkAreas[SyncTime.AFTER_START_UP]
           OF
             // NO_SYNCHRONIZATION
             SyncMode.NO_SYNCHRONIZATION : ; // no further action

             // CLIENT_TO_SERVER
             SyncMode.CLIENT_TO_SERVER :
               // set timeout
               SetTimeout(PT := _rTimeout, rTimer := _rTimer);
               // inc step counter
              _rStep := 11;

             // SERVER_TO_CLIENT
             SyncMode.SERVER_TO_CLIENT :
               // set timeout
               SetTimeout(PT := _rTimeout, rTimer := _rTimer);
               // inc step counter
              _rStep := 12;

             // AUTOMATIC
             SyncMode.AUTOMATIC :
               // set timeout
               SetTimeout(PT := _rTimeout, rTimer := _rTimer);
               // inc step counter
              _rStep := 13;
           END_CASE
         ELSE
           // datas changeḍ on both sides ? -> Warning
           IF (( NOT AxesGroup.State.SyncStatePlc.InSync.WorkArea ) AND
               ( NOT AxesGroup.State.SyncStateRc .InSync.WorkArea ))
           THEN
             WarningID := RobotLibraryWarningIdEnum.WARN_WORK_AREA_SYNC_BOTH_SIDES_CHANGED;
           END_IF
         END_IF

    // ------------------------------------------
    // SyncMode : CLIENT_TO_SERVER
    // ------------------------------------------
    11 : // Conflict triggerd by PLC ?
         IF ( NOT AxesGroup.State.SyncStatePlc.InSync.WorkArea )
         THEN
           // search for changed index
           FOR _rSyncIdx := 0 TO AxesGroup.State.UnifiedWorkAreaIndex
           DO
             IF ( AxesGroup.State.DataChanged.WorkArea[_rSyncIdx] )
             THEN
               // set timeout
               SetTimeout(PT := _rTimeout, rTimer := _rTimer);
               // inc step counter
              _rStep := 30; // -> write PLC data to RC
               EXIT;
  					 END_IF
           END_FOR

           // Create log entry
           CreateLogMessagePara3 ( Timestamp   := SystemTime,
                                   MessageType := MessageType.CMD,
                                   Severity    := Severity.DEBUG,
                                   MessageCode := 0,
                                   MessageText := 'SyncWorkArea: Synchronization of WorkArea[{1}] triggered by PLC, SyncMode = {2}, SyncTime = {3}, SyncDirection = PLC -> RC',
                                   Para1       :=  DINT_TO_STRING(_rSyncIdx),
                                   Para2       :=  SYNC_MODE_TO_STRING(AxesGroup.Parameter.Plc.Parameter.SynchronizationModes.WorkAreas[SyncTime.AFTER_START_UP]),
                                   Para3       :=  SYNC_TIME_TO_STRING(SyncTime.AFTER_START_UP));
                                   RETURN;
         END_IF

         // Conflict triggered by RC ?
         IF ( NOT AxesGroup.State.SyncStateRc.InSync.WorkArea )
         THEN
           // get changed index
          _rSyncIdx :=  LIMIT(0, AxesGroup.State.SyncStateRc.UnSyncNo.WorkArea, AxesGroup.State.UnifiedWorkAreaIndex);
           // set timeout
           SetTimeout(PT := _rTimeout, rTimer := _rTimer);
           // inc step counter
          _rStep := 30; // -> write PLC data to RC

           // Create log entry
           CreateLogMessagePara3 ( Timestamp   := SystemTime,
                                   MessageType := MessageType.CMD,
                                   Severity    := Severity.DEBUG,
                                   MessageCode := 0,
                                   MessageText := 'SyncWorkArea: Synchronization of WorkArea[{1}] triggered by RC, SyncMode = {2}, SyncTime = {3}, SyncDirection = PLC -> RC',
                                   Para1       :=  DINT_TO_STRING(_rSyncIdx),
                                   Para2       :=  SYNC_MODE_TO_STRING(AxesGroup.Parameter.Plc.Parameter.SynchronizationModes.WorkAreas[SyncTime.AFTER_START_UP]),
                                   Para3       :=  SYNC_TIME_TO_STRING(SyncTime.AFTER_START_UP));
                                   RETURN;
  			 END_IF

         // set timeout
         SetTimeout(PT := _rTimeout, rTimer := _rTimer);
         // jump back
        _rStep := 10;

    // ------------------------------------------
    // SyncMode : SERVER_TO_CLIENT
    // ------------------------------------------
    12 : // Conflict triggerd by PLC ?
         IF ( NOT AxesGroup.State.SyncStatePlc.InSync.WorkArea )
         THEN
           // search for changed index
           FOR _rSyncIdx := 0 TO AxesGroup.State.UnifiedWorkAreaIndex
           DO
             IF ( AxesGroup.State.DataChanged.WorkArea[_rSyncIdx] )
             THEN
               // set timeout
               SetTimeout(PT := _rTimeout, rTimer := _rTimer);
               // inc step counter
              _rStep := 20; // -> read RC data and write it to PLC
               EXIT;
  					 END_IF
           END_FOR

           // Create log entry
           CreateLogMessagePara3 ( Timestamp   := SystemTime,
                                   MessageType := MessageType.CMD,
                                   Severity    := Severity.DEBUG,
                                   MessageCode := 0,
                                   MessageText := 'SyncWorkArea: Synchronization of WorkArea[{1}] triggered by PLC, SyncMode = {2}, SyncTime = {3}, SyncDirection = RC -> PLC',
                                   Para1       :=  DINT_TO_STRING(_rSyncIdx),
                                   Para2       :=  SYNC_MODE_TO_STRING(AxesGroup.Parameter.Plc.Parameter.SynchronizationModes.WorkAreas[SyncTime.AFTER_START_UP]),
                                   Para3       :=  SYNC_TIME_TO_STRING(SyncTime.AFTER_START_UP));
                                   RETURN;
         END_IF

         // Conflict triggered by RC ?
         IF ( NOT AxesGroup.State.SyncStateRc.InSync.WorkArea )
         THEN
           // get changed index
          _rSyncIdx := LIMIT(0, AxesGroup.State.SyncStateRc.UnSyncNo.WorkArea, AxesGroup.State.UnifiedWorkAreaIndex);
           // set timeout
           SetTimeout(PT := _rTimeout, rTimer := _rTimer);
           // inc step counter
          _rStep := 20; // -> read RC data and write it to PLC

           // Create log entry
           CreateLogMessagePara3 ( Timestamp   := SystemTime,
                                   MessageType := MessageType.CMD,
                                   Severity    := Severity.DEBUG,
                                   MessageCode := 0,
                                   MessageText := 'SyncWorkArea: Synchronization of WorkArea[{1}] triggered by RC, SyncMode = {2}, SyncTime = {3}, SyncDirection = RC -> PLC',
                                   Para1       :=  DINT_TO_STRING(_rSyncIdx),
                                   Para2       :=  SYNC_MODE_TO_STRING(AxesGroup.Parameter.Plc.Parameter.SynchronizationModes.WorkAreas[SyncTime.AFTER_START_UP]),
                                   Para3       :=  SYNC_TIME_TO_STRING(SyncTime.AFTER_START_UP));
                                   RETURN;
  			 END_IF

         // set timeout
         SetTimeout(PT := _rTimeout, rTimer := _rTimer);
         // jump back
        _rStep := 10;

    // ------------------------------------------
    // SyncMode : AUTOMATIC
    // ------------------------------------------
    13 : // Conflict triggerd by PLC ?
         IF ( NOT AxesGroup.State.SyncStatePlc.InSync.WorkArea )
         THEN
           // search for changed index
           FOR _rSyncIdx := 0 TO AxesGroup.State.UnifiedWorkAreaIndex
           DO
             IF ( AxesGroup.State.DataChanged.WorkArea[_rSyncIdx] )
             THEN
               // set timeout
               SetTimeout(PT := _rTimeout, rTimer := _rTimer);
               // inc step counter
              _rStep := 30; // -> write PLC data to RC
               EXIT;
  					 END_IF
           END_FOR

           // Create log entry
           CreateLogMessagePara3 ( Timestamp   := SystemTime,
                                   MessageType := MessageType.CMD,
                                   Severity    := Severity.DEBUG,
                                   MessageCode := 0,
                                   MessageText := 'SyncWorkArea: Synchronization of WorkArea[{1}] triggered by PLC, SyncMode = {2}, SyncTime = {3}, SyncDirection = PLC -> RC',
                                   Para1       :=  DINT_TO_STRING(_rSyncIdx),
                                   Para2       :=  SYNC_MODE_TO_STRING(AxesGroup.Parameter.Plc.Parameter.SynchronizationModes.WorkAreas[SyncTime.AFTER_START_UP]),
                                   Para3       :=  SYNC_TIME_TO_STRING(SyncTime.AFTER_START_UP));
                                   RETURN;
         END_IF

         // Conflict triggered by RC ?
         IF ( NOT AxesGroup.State.SyncStateRc.InSync.WorkArea )
         THEN
           // get changed index
          _rSyncIdx := LIMIT(0, AxesGroup.State.SyncStateRc.UnSyncNo.WorkArea, AxesGroup.State.UnifiedWorkAreaIndex);
           // set timeout
           SetTimeout(PT := _rTimeout, rTimer := _rTimer);
           // inc step counter
          _rStep := 20; // -> read RC data an write it to PLC

           // Create log entry
           CreateLogMessagePara3 ( Timestamp   := SystemTime,
                                   MessageType := MessageType.CMD,
                                   Severity    := Severity.DEBUG,
                                   MessageCode := 0,
                                   MessageText := 'SyncWorkArea: Synchronization of WorkArea[{1}] triggered by RC, SyncMode = {2}, SyncTime = {3}, SyncDirection = RC -> PLC',
                                   Para1       :=  DINT_TO_STRING(_rSyncIdx),
                                   Para2       :=  SYNC_MODE_TO_STRING(AxesGroup.Parameter.Plc.Parameter.SynchronizationModes.WorkAreas[SyncTime.AFTER_START_UP]),
                                   Para3       :=  SYNC_TIME_TO_STRING(SyncTime.AFTER_START_UP));
                                   RETURN;
  			 END_IF

         // set timeout
         SetTimeout(PT := _rTimeout, rTimer := _rTimer);
         // jump back
        //_rStep := 10;

    // ------------------------------------------
    // Read Data from RC and write it to PLC
    // ------------------------------------------
    20 : IF (( NOT _readWorkArea.Busy  ) AND
             ( NOT _readWorkArea.Error ))
         THEN
           // set command parameter
          _readWorkArea.ParCmd.WorkAreaNo := _rSyncIdx;
           // execute command
          _readWorkArea.Execute := TRUE;
           // set timeout
           SetTimeout(PT := _rTimeout, rTimer := _rTimer);
           // inc step counter
          _rStep := _rStep + 1;
         ELSE
           // check error ?
           IF (_readWorkArea.Error)
           THEN
             ErrorID     := _readWorkArea.ErrorID;
             ErrorAddTxt := _readWorkArea.ErrorAddTxt;
           END_IF

           // timeout exceeded ?
           IF (CheckTimeout(_rTimer) = RobotLibraryConstants.OK)
           THEN
             ErrorID     := RobotLibraryErrorIdEnum.ERR_TIMEOUT_CMD;
             ErrorAddTxt := CONCAT(_stepName, DINT_TO_STRING(_rStep));
           END_IF
         END_IF

    21 : IF (( NOT _readWorkArea.Busy  ) AND
             ( NOT _readWorkArea.Error ) AND
             (     _readWorkArea.Done  ))
         THEN
           // reset execution
          _readWorkArea.Execute := FALSE;
           // update internal WorkArea data
           WorkAreas[_rSyncIdx].Data := _readWorkArea.OutCmd.WorkAreaData;
          _workAreas[_rSyncIdx].Data := _readWorkArea.OutCmd.WorkAreaData;
           // set available bit
           WorkAreas[_rSyncIdx].Available := TRUE;
          _workAreas[_rSyncIdx].Available := TRUE;
           // set timeout
           SetTimeout(PT := _rTimeout, rTimer := _rTimer);
           // inc step counter
          _rStep := 10; // -> jump to after startup
         ELSE
           // check error ?
           IF (_readWorkArea.Error)
           THEN
             ErrorID     := _readWorkArea.ErrorID;
             ErrorAddTxt := _readWorkArea.ErrorAddTxt;
             // reset available bit
             WorkAreas[_rSyncIdx].Available := FALSE;
            _workAreas[_rSyncIdx].Available := FALSE;
           END_IF

           // timeout exceeded ?
           IF (CheckTimeout(_rTimer) = RobotLibraryConstants.OK)
           THEN
             ErrorID     := RobotLibraryErrorIdEnum.ERR_TIMEOUT_CMD;
             ErrorAddTxt := CONCAT(_stepName, DINT_TO_STRING(_rStep));
           END_IF
         END_IF

    // ------------------------------------------
    // Write data from PLC to RC
    // ------------------------------------------
    30 : IF (( NOT _writeWorkArea.Busy  ) AND
             ( NOT _writeWorkArea.Error ))
         THEN
           // set command parameter
          _writeWorkArea.ParCmd.WorkAreaNo   := _rSyncIdx;
          _writeWorkArea.ParCmd.WorkAreaData :=  WorkAreas[_rSyncIdx].Data;
           // execute command
          _writeWorkArea.Execute := TRUE;
           // set timeout
           SetTimeout(PT := _rTimeout, rTimer := _rTimer);
           // inc step counter
          _rStep := _rStep + 1;
         ELSE
           // check error ?
           IF (_writeWorkArea.Error)
           THEN
             ErrorID     := _writeWorkArea.ErrorID;
             ErrorAddTxt := _writeWorkArea.ErrorAddTxt;;
           END_IF

           // timeout exceeded ?
           IF (CheckTimeout(_rTimer) = RobotLibraryConstants.OK)
           THEN
             ErrorID     := RobotLibraryErrorIdEnum.ERR_TIMEOUT_CMD;
             ErrorAddTxt := CONCAT(_stepName, DINT_TO_STRING(_rStep));
           END_IF
         END_IF

    31 : IF (( NOT _writeWorkArea.Busy  ) AND
             ( NOT _writeWorkArea.Error ) AND
             (     _writeWorkArea.Done  ))
         THEN
           // execute command
          _writeWorkArea.Execute := FALSE;
           // update internal WorkArea data
          _workAreas[_rSyncIdx] := WorkAreas[_rSyncIdx];
           // set available bit
           WorkAreas[_rSyncIdx].Available := TRUE;
          _workAreas[_rSyncIdx].Available := TRUE;
           // set timeout
           SetTimeout(PT := _rTimeout, rTimer := _rTimer);
           // inc step counter
          _rStep := 10; // -> jump to after startup;
         ELSE
           // check error ?
           IF (_writeWorkArea.Error)
           THEN
             WarningID := RobotLibraryWarningIdEnum.WARN_WORK_AREA_SYNC_FAILED_BY_ERROR_OF_READ_OR_WRITE_CMD;
             // reset available bit
             WorkAreas[_rSyncIdx].Available := FALSE;
            _workAreas[_rSyncIdx].Available := FALSE;
           END_IF

           // timeout exceeded ?
           IF (CheckTimeout(_rTimer) = RobotLibraryConstants.OK)
           THEN
             ErrorID     := RobotLibraryErrorIdEnum.ERR_TIMEOUT_CMD;
             ErrorAddTxt := CONCAT(_stepName, DINT_TO_STRING(_rStep));
           END_IF
         END_IF

  ELSE
    // invalid step
    ErrorID     := RobotLibraryErrorIdEnum.ERR_INVALID_STEP;
    ErrorAddTxt := CONCAT(_stepName , DINT_TO_STRING(_stepCmd));
  END_CASE

END_METHOD

METHOD PRIVATE HandleTelegramStateCtrl
VAR_INPUT
END_VAR

  // Telegram Control
  // ----------------
  IF ( _lastTelegramControl <> GetHalfeByteLo(Telegram.PlcToRob.Header.AxesGroupID_Control))
  THEN
    // Create log entry
    CreateLogMessagePara2 ( Timestamp   := SystemTime,
                            MessageType := MessageType.CMD,
                            Severity    := Severity.INFO,
                            MessageCode := 0,
                            MessageText := 'SRCI Interface control changed from {1} to {2}',
                            Para1       := TELEGRAM_CONTROL_TO_STRING(_lastTelegramControl),
                            Para2       := TELEGRAM_CONTROL_TO_STRING(GetHalfeByteLo(Telegram.PlcToRob.Header.AxesGroupID_Control)));

    _lastTelegramControl := GetHalfeByteLo(Telegram.PlcToRob.Header.AxesGroupID_Control);
  END_IF

  // Telegram State
  // ----------------
  IF ( _lastTelegramState <> Telegram.RobToPlc.Header.TelegramState)
  THEN
    // Create log entry
    CreateLogMessagePara2 ( Timestamp   := SystemTime,
                            MessageType := MessageType.CMD,
                            Severity    := Severity.INFO,
                            MessageCode := 0,
                            MessageText := 'SRCI Interface state changed from {1} to {2}',
                            Para1       := TELEGRAM_STATE_TO_STRING(_lastTelegramState),
                            Para2       := TELEGRAM_STATE_TO_STRING(Telegram.RobToPlc.Header.TelegramState));

    _lastTelegramState := Telegram.RobToPlc.Header.TelegramState;
  END_IF

END_METHOD

METHOD HandleUserData
VAR_IN_OUT
   /// Robot assignment of function
  AxesGroup    : AxesGroup;
  ///  User data stored on the PLC according to Table 6-10
  UserData     : UserData;
END_VAR

  // Common
  UserData.LogLevel                          := LogLevel;

  UserData.PLCManufacturedID                 := _parCfg.Plc.Parameter.ManufacturedID;
  UserData.PLCOrderID                        := _parCfg.Plc.Parameter.OrderID;
  UserData.PLCSerialNumber                   := _parCfg.Plc.Parameter.SerialNumber;
  UserData.PLCFirmwareVersion                := _parCfg.Plc.Parameter.FirmwareVersion;
  UserData.PLCInterfaceVersion               := _parCfg.Plc.Parameter.InterfaceVersion;
  UserData.PLCLibraryVersion                 :=  RobotLibraryConstants.PLCLibraryVersion;

  // Communication
  UserData.LifeSignTimeOut                   := _parCfg.Com.LifeSignTimeOut;

  // Plc Parameter
  UserData.SynchronizationModes              := _parCfg.Plc.Parameter.SynchronizationModes;
  UserData.EnableSync                        :=  SyncModesToDataEnableSync(Value := _parCfg.Plc.Parameter.SynchronizationModes);

  // Robot Parameter
  UserData.DelayTime                         := _parCfg.Rob.Parameter.DelayTime;
  UserData.WaitForNrOfCmd                    := _parCfg.Rob.Parameter.WaitForNrOfCmd;
  UserData.WaitAtBlendingZone                := _parCfg.Rob.Parameter.WaitAtBlendingZone;
  UserData.AllowSecSeqWhileSubprogram        := _parCfg.Rob.Parameter.AllowSecSeqWhileSubprogram;
  UserData.AllowDynamicBlending              := _parCfg.Rob.Parameter.AllowDynamicBlending;
  UserData.SyncReaction                      := _parCfg.Rob.Parameter.SyncReaction;
  UserData.SyncDelay                         := _parCfg.Rob.Parameter.SyncDelay;
  UserData.MessageLevel                      := _parcfg.Rob.Parameter.MessageLevel;

  // ReadRobotData
  UserData.RCManufacturer                    := AxesGroup.State.RobotData.RCManufacturer;
  UserData.RCOrderID                         := AxesGroup.State.RobotData.RCOrderID;
  UserData.RCSerialNumber                    := AxesGroup.State.RobotData.RCSerialNumber;
  UserData.RASerialNumber                    := AxesGroup.State.RobotData.RASerialNumber;
  UserData.RCFirmwareVersion                 := AxesGroup.State.RobotData.RCFirmwareVersion;

  UserData.RCInterpreterVersion.MajorVersion := STRING_TO_USINT(MID(AxesGroup.State.RobotData.RCInterpreterVersion, LEN := 1, POS := 1));
  UserData.RCInterpreterVersion.MinorVersion := STRING_TO_USINT(MID(AxesGroup.State.RobotData.RCInterpreterVersion, LEN := 1, POS := 2));
  UserData.RCInterpreterVersion.PatchVersion := STRING_TO_USINT(MID(AxesGroup.State.RobotData.RCInterpreterVersion, LEN := 1, POS := 3));

  UserData.AxisJointUsed                     := AxesGroup.State.RobotData.AxisJointUsed;
  UserData.AxisExternalUsed                  := AxesGroup.State.RobotData.AxisExternalUsed;
  UserData.AxisJointUnit                     := AxesGroup.State.RobotData.AxisJointUnit;
  UserData.AxisExternalUnit                  := AxesGroup.State.RobotData.AxisExternalUnit;
  UserData.RCSupportedFunctions              := AxesGroup.State.RobotData.RCSupportedFunctions;

  UserData.BrakeTestRequired                 := AxesGroup.State.ConfigurationData.BrakeTestRequired;
  UserData.PathAccuracyMode                  := AxesGroup.State.ConfigurationData.PathAccuracyMode;
  UserData.AvoidSingularity                  := AxesGroup.State.ConfigurationData.AvoidSingularity;
  UserData.ConstantVelocitySupported         := AxesGroup.State.ConfigurationData.ConstantVelocitySupported;
  UserData.StepModeExactStopActive           := AxesGroup.State.ConfigurationData.StepModeExactStopActive;
  UserData.StepModeBlendingActive            := AxesGroup.State.ConfigurationData.StepModeBlendingActive;
  UserData.AcceleratingSupported             := AxesGroup.State.ConfigurationData.AcceleratingSupported;
  UserData.DeceleratingSupported             := AxesGroup.State.ConfigurationData.DecceleratingSupported;

  UserData.Initialized                       := Initialized;
  UserData.Synchronized                      := Synchronized;

  // Cyclic data
  UserData.RCSRCIVersion                     := AxesGroup.Cyclic.RobToPlc.SRCIVersion;
  UserData.IsMoving                          := AxesGroup.Cyclic.RobToPlc.StatusRobotArm.IsMoving;
  UserData.PrimarySequencePaused             := AxesGroup.Cyclic.RobToPlc.StatusRobotArm.PrimarySequencePaused;
  UserData.InPrimaryPos                      := AxesGroup.Cyclic.RobToPlc.StatusRobotArm.InPrimaryPos;
  UserData.SecondarySequenceActive           := AxesGroup.Cyclic.RobToPlc.StatusRobotArm.SecondarySequenceActive;
  UserData.ErrorPending                      := AxesGroup.Cyclic.RobToPlc.StatusRobotArm.ErrorPending;
  UserData.RestartInProgress                 := AxesGroup.Cyclic.RobToPlc.StatusRobotArm.RestartInProgress;
  UserData.Enabled                           := AxesGroup.Cyclic.RobToPlc.StatusRobotArm.Enabled;
  UserData.Idle                              := AxesGroup.Cyclic.RobToPlc.StatusRobotArm.RaSequenceState = RaSequenceState.IDLE;
  UserData.Executing                         := AxesGroup.Cyclic.RobToPlc.StatusRobotArm.RaSequenceState = RaSequenceState.EXECUTING;
  UserData.Interrupted                       := AxesGroup.Cyclic.RobToPlc.StatusRobotArm.RaSequenceState = RaSequenceState.INTERRUPTED;
  UserData.IsBlending                        := AxesGroup.Cyclic.RobToPlc.StatusRobotArm.IsBlending;
  UserData.OperationMode                     := AxesGroup.Cyclic.RobToPlc.StatusRobotArm.OperationMode;
  UserData.CollisionDetectionEnabled         := AxesGroup.Cyclic.RobToPlc.StatusRobotArm.CollisionDetectedEnabled;
  UserData.CollisionDetected                 := AxesGroup.Cyclic.RobToPlc.StatusRobotArm.CollisionDetected;
  UserData.RestartRequested                  := AxesGroup.Cyclic.RobToPlc.StatusRobotArm.RestartRequested;
  UserData.Accelerating                      := AxesGroup.Cyclic.RobToPlc.StatusRobotArm.Accelerating;
  UserData.Decelerating                      := AxesGroup.Cyclic.RobToPlc.StatusRobotArm.Decelerating;
  UserData.ConstantVelocity                  := AxesGroup.Cyclic.RobToPlc.StatusRobotArm.ConstantVelocity;
  UserData.ActualOverride                    := PERCENT_UINT_TO_REAL( Value := AxesGroup.Cyclic.RobToPlc.Override, IsOptional := FALSE);

  // Cyclic optional data
  UserData.CartesianPosition                 := AxesGroup.CyclicOptional.RobToPlc.CartesianPosition;
  UserData.ExtCartesianPosition              := AxesGroup.CyclicOptional.RobToPlc.CartesianPositionExt;
  UserData.JointPosition                     := AxesGroup.CyclicOptional.RobToPlc.JointPosition;
  UserData.ExtJointPosition                  := AxesGroup.CyclicOptional.RobToPlc.JointPositionExt;

  // Synchronizing
  UserData.ToolDataSynchronizing             := AxesGroup.State.Synchronizing.Tool;
  UserData.FrameDataSynchronizing            := AxesGroup.State.Synchronizing.Frame;
  UserData.LoadDataSynchronizing             := AxesGroup.State.Synchronizing.Load;
  UserData.WorkAreaDataSynchronizing         := AxesGroup.State.Synchronizing.WorkAreas;
  UserData.SWLimitsSynchronizing             := AxesGroup.State.Synchronizing.SwLimits;
  UserData.DefaultDynamicsSynchronizing      := AxesGroup.State.Synchronizing.DefaultDynamics;
  UserData.ReferenceDynamicsSynchronizing    := AxesGroup.State.Synchronizing.ReferenceDynamics;

  UserData.ActivateTwoSequences              := _parCfg.Com.TwoSequences;
  UserData.ReadingCartesianPosition          :=  AxesGroup.State.ReadingCartesianPosition;
  UserData.ReadingExtCartesianPosition       :=  AxesGroup.State.ReadingCartesianPositionExt;
  UserData.ReadingJointPosition              :=  AxesGroup.State.ReadingJointPosition;
  UserData.ReadingExtJointPosition           :=  AxesGroup.State.ReadingJointPositionExt;

END_METHOD

METHOD PRIVATE OnCall
VAR_IN_OUT
   /// Robot assignment of function
  AxesGroup : AxesGroup;
END_VAR

  // map numeric value to enum, so that the corresponding message text is directly shown by the tooltip
  ErrorIdEnum   := ErrorId;
  WarningIdEnum := WarningId;
  InfoIdEnum    := InfoId;

  Error := ErrorID <> RobotLibraryConstants.OK ;

  // Check Payload and In/Out data size
  IF (( RobotLibraryParameter.ROBOT_IN_DATA_MAX  < 64 ) OR
      ( RobotLibraryParameter.ROBOT_OUT_DATA_MAX < 64 ))
  THEN
    ErrorID := RobotLibraryErrorIdEnum.ERR_INVALID_LIBRARY_PARA;
    RETURN;
  END_IF

  // Check AxesGroupID valid
  IF (( AxesGroupID < RobotLibraryConstants.AXES_GROUP_ID_MIN ) OR
      ( AxesGroupID > RobotLibraryConstants.AXES_GROUP_ID_MAX ))
  THEN
    ErrorID := RobotLibraryErrorIdEnum.ERR_INVALID_AXES_GROUP_ID;
    RETURN;
  END_IF

  // Reset flag for initialization / Synchronization
  IF ( Initialized OR Synchronized) AND ( AxesGroup.Cyclic.RobToPlc.TelegramState <> TelegramState.INITIALIZED)
  THEN
    // Reset initialized flag
    Initialized := FALSE;
    // Reset Synchronized flag
    Synchronized := FALSE;
    // Set error
    ErrorID := RobotLibraryErrorIdEnum.ERR_INIT_LOST_UNKNOWN_0x80A2;
  END_IF

  // Warning for ACR Registers running low
  IF ( AxesGroup.Acyclic.ActiveCommandRegister.CurrentAcrUsagePercent > RobotLibraryParameter.ACR_USAGE_WARNING_LIMIT )
  THEN
    WarningID := RobotLibraryWarningIdEnum.WARN_ACR_FREE_ENTRIES_LOW;
  END_IF

  // Check configuration parameter changed ?
  CheckParameterChanged(AxesGroup := AxesGroup);

END_METHOD

METHOD OnExecRun : DINT
VAR_IN_OUT
  /// Robot assignment of function
  AxesGroup         : AxesGroup;
END_VAR

  // building rising and falling edges
  _enable_R( CLK := Enable);
  _enable_F( CLK := Enable);

  IF ( _enable_F.Q)
  THEN
    Reset(AxesGroup := AxesGroup);
  END_IF

  OnExecRun := RobotLibraryConstants.RUNNING;

  CASE _stepCmd OF

    00:  IF ( _enable_R.Q )
         THEN
           // Create log entry
           CreateLogMessage ( Timestamp   := SystemTime,
                              MessageType := MessageType.CMD,
                              Severity    := Severity.INFO,
                              MessageCode := 0,
                              MessageText := 'Robot Task Enabled');

           // reset the rising edge
          _enable_R();
           // set busy flag
           Busy := TRUE;
           // set timeout
           SetTimeout(PT := _timeoutCmd, rTimer := _timerCmd);
           // Reset FastStop
           AxesGroup.Cyclic.PlcToRob.FastStop := 0;
           // Reset Active command register
           AxesGroup.Acyclic.ActiveCommandRegister.Reset();

           // check parameter valid
           IF ( CheckParameterValid(AxesGroup := AxesGroup) )
           THEN
             // take configuration parameter if not yet enabled
            _parCfg := ParCfg;
             // inc step counter
            _stepCmd := _stepCmd + 1;
           END_IF
         END_IF

    01:  CASE AxesGroup.Cyclic.RobToPlc.TelegramState  OF

           TelegramState.UNDEFINED : ;

           TelegramState.ERROR_161_TELEGRAM_CONTROL_MISMATCH_TELEGRAM_STATE..TelegramState.ERROR_172_TELEGRAM_NUMBER_NOT_SUPPORTED:

             // clear error
             AxesGroup.Cyclic.PlcToRob.Control := ControlHalfByte.ACK_ERROR;
             AxesGroup.Cyclic.PlcToRob.Control := ControlHalfByte.RESET; // always a reset, so that on the robot side the ACR is reseted

           TelegramState.ERROR_173_SERVER_CONNECTION_LOST:

             // Reset interface including the ACR register on server side
             AxesGroup.Cyclic.PlcToRob.Control := ControlHalfByte.RESET;

           TelegramState.READY_TO_RESUME :

             // Resume
             AxesGroup.Cyclic.PlcToRob.Control := ControlHalfByte.RESUME;

           TelegramState.READY_FOR_INITIALIZATION:

             // Request initialization
             AxesGroup.Cyclic.PlcToRob.Control := ControlHalfByte.INITIALIZE;

           TelegramState.INITIALIZED:

             // Reset Telegram Control
             AxesGroup.Cyclic.PlcToRob.Control := ControlHalfByte.NONE;

             // Check SRCI Version is compatible ?
             IF ( AxesGroup.Cyclic.RobToPlc.SRCIVersion.MajorVersion = RobotLibraryConstants.SRCIVersion.MajorVersion )
             THEN
               // set timeout
               SetTimeout(PT := _timeoutCmd, rTimer := _timerCmd);
               // inc step counter
              _stepCmd := _stepCmd + 1;
             ELSE
               // set error
               ErrorID     := RobotLibraryErrorIdEnum.ERR_SRCI_MAJOR_VERSION_INCOMPATIBLE_0x80A4;
               ErrorAddTxt := CONCAT('_stepCmd = ' , DINT_TO_STRING(_stepCmd));
             END_IF

         ELSE
           // TelegrammState in error
           ErrorID := RobotLibraryErrorIdEnum.ERR_INIT_LOST_UNKNOWN_0xA2;
           ErrorAddTxt := CONCAT('_stepCmd = ' , DINT_TO_STRING(_stepCmd));
         END_CASE

         // timeout exceeded ?
         IF (CheckTimeout(_timerCmd) = RobotLibraryConstants.OK)
         THEN
           // Check Telegram State error ?
           IF (( AxesGroup.Cyclic.RobToPlc.TelegramState >= TelegramState.ERROR_161_TELEGRAM_CONTROL_MISMATCH_TELEGRAM_STATE ) OR
               ( AxesGroup.Cyclic.RobToPlc.TelegramState <= TelegramState.ERROR_173_SERVER_CONNECTION_LOST                   ))
           THEN
             ErrorID     := AxesGroup.Cyclic.RobToPlc.TelegramState;
             ErrorAddTxt := CONCAT('_stepCmd = ' , DINT_TO_STRING(_stepCmd));
           ELSE
             ErrorID     := RobotLibraryErrorIdEnum.ERR_TIMEOUT_CMD;
             ErrorAddTxt := CONCAT('_stepCmd = ' , DINT_TO_STRING(_stepCmd));
           END_IF
         END_IF

    02: IF (( NOT _readMessages.Busy  ) AND
            ( NOT _readMessages.Error ))
        THEN
          // start function block
         _readMessages.Enable := TRUE;
         _readMessages.ParCmd.MsgID := 0;
         _readMessages.ParCmd.MessageLevel := _parCfg.Rob.Parameter.MessageLevel;

          // set timeout
          SetTimeout(PT := _timeoutCmd, rTimer := _timerCmd);
          // inc step counter
         _stepCmd := _stepCmd + 1;
        ELSE
          // check error ?
          IF (_readMessages.Error)
          THEN
            ErrorID     := _readMessages.ErrorID;
            ErrorAddTxt := _readMessages.ErrorAddTxt;;
          END_IF
          // timeout exceeded ?
          IF (CheckTimeout(_timerCmd) = RobotLibraryConstants.OK)
          THEN
            ErrorID     := RobotLibraryErrorIdEnum.ERR_TIMEOUT_CMD;
            ErrorAddTxt := CONCAT('_stepCmd = ' , DINT_TO_STRING(_stepCmd));
          END_IF
        END_IF

    03: IF ((     _readMessages.Enabled ) AND
            ( NOT _readMessages.Busy    ) AND
            ( NOT _readMessages.Error   ))
        THEN
          // ---------------------------------------------------------------
          // !!! ReadMessages must stay active for the Message mechanism !!!
          // ---------------------------------------------------------------
          // ReadMessages.Enable := FALSE;
          // set timeout
          SetTimeout(PT := _timeoutCmd, rTimer := _timerCmd);
          // inc step counter
         _stepCmd := _stepCmd + 1;
        ELSE
           // check error ?
           IF (_readMessages.Error)
           THEN
             ErrorID     := _readMessages.ErrorID;
             ErrorAddTxt := _readMessages.ErrorAddTxt;;
           END_IF

           // timeout exceeded ?
           IF (CheckTimeout(_timerCmd) = RobotLibraryConstants.OK)
           THEN
             ErrorID     := RobotLibraryErrorIdEnum.ERR_TIMEOUT_CMD;
             ErrorAddTxt := CONCAT('_stepCmd = ' , DINT_TO_STRING(_stepCmd));
           END_IF
         END_IF

    04: IF (( NOT _exchangeConfiguration.Busy  ) AND
            ( NOT _exchangeConfiguration.Error ))
        THEN
          // set command parameter
         _exchangeConfiguration.ParCmd.LogLevel                           :=  LogLevel;
         _exchangeConfiguration.ParCmd.WaitAtBlendingZone                 := _parCfg.Rob.Parameter.WaitAtBlendingZone;
         _exchangeConfiguration.ParCmd.AllowSecSeqWhileSubprogram         := _parCfg.Rob.Parameter.AllowSecSeqWhileSubprogram;
         _exchangeConfiguration.ParCmd.AllowDynamicBlending               := _parCfg.Rob.Parameter.AllowDynamicBlending;
         _exchangeConfiguration.ParCmd.DelayTime                          := _parCfg.Rob.Parameter.DelayTime;
         _exchangeConfiguration.ParCmd.WaitForNrOfCmd                     := _parCfg.Rob.Parameter.WaitForNrOfCmd;
         _exchangeConfiguration.ParCmd.LifeSignTimeOut                    :=  TIME_TO_UINT(_parCfg.Com.LifeSignTimeOut);
         _exchangeConfiguration.ParCmd.SyncDelay                          := _parCfg.Rob.Parameter.SyncDelay;
         _exchangeConfiguration.ParCmd.SyncReaction                       := _parCfg.Rob.Parameter.SyncReaction;
         _exchangeConfiguration.ParCmd.DataEnableSync                     :=  SyncModesToDataEnableSync(Value := _parCfg.Plc.Parameter.SynchronizationModes);
         _exchangeConfiguration.ParCmd.DataInSync.ToolsInSync             :=  FALSE;
         _exchangeConfiguration.ParCmd.DataInSync.FramesInSync            :=  FALSE;
         _exchangeConfiguration.ParCmd.DataInSync.LoadsInSync             :=  FALSE;
         _exchangeConfiguration.ParCmd.DataInSync.WorkAreasInSync         :=  FALSE;
         _exchangeConfiguration.ParCmd.DataInSync.SoftwareLimitsInSync    :=  FALSE;
         _exchangeConfiguration.ParCmd.DataInSync.DefaultDynamicsInSync   :=  FALSE;
         _exchangeConfiguration.ParCmd.DataInSync.ReferenceDynamicsInSync :=  FALSE;

          // start function block
         _exchangeConfiguration.Enable := TRUE;
          // set timeout
          SetTimeout(PT := _timeoutCmd, rTimer := _timerCmd);
          // inc step counter
         _stepCmd := _stepCmd + 1;
        ELSE
          // check error ?
          IF (_exchangeConfiguration.Error)
          THEN
            ErrorID     := _exchangeConfiguration.ErrorID;
            ErrorAddTxt := _exchangeConfiguration.ErrorAddTxt;;
          END_IF

          // timeout exceeded ?
          IF (CheckTimeout(_timerCmd) = RobotLibraryConstants.OK)
          THEN
            ErrorID     := RobotLibraryErrorIdEnum.ERR_TIMEOUT_CMD;
            ErrorAddTxt := CONCAT('_stepCmd = ' , DINT_TO_STRING(_stepCmd));
          END_IF
        END_IF

    05: IF (( NOT _exchangeConfiguration.Busy    ) AND
            (     _exchangeConfiguration.Enabled ))
        THEN
          // ---------------------------------------------------------------------
          // !!! ExchangeConfiguration must stay active for the Sync mechanism !!!
          // ---------------------------------------------------------------------
          // ExchangeConfiguration.Enable := FALSE;
          // set timeout
          SetTimeout(PT := _timeoutCmd, rTimer := _timerCmd);
          // inc step counter
         _stepCmd := _stepCmd + 1;
        ELSE
          // check error ?
          IF (_exchangeConfiguration.Error)
          THEN
            ErrorID     := _exchangeConfiguration.ErrorID;
            ErrorAddTxt := _exchangeConfiguration.ErrorAddTxt;;
          END_IF

          // timeout exceeded ?
          IF (CheckTimeout(_timerCmd) = RobotLibraryConstants.OK)
          THEN
            ErrorID     := RobotLibraryErrorIdEnum.ERR_TIMEOUT_CMD;
            ErrorAddTxt := CONCAT('_stepCmd = ' , DINT_TO_STRING(_stepCmd));
          END_IF
        END_IF

    06: IF (( NOT _readRobotData.Busy  ) AND
            ( NOT _readRobotData.Error ))
        THEN
          // start function block
         _readRobotData.Execute := TRUE;
          // set timeout
          SetTimeout(PT := _timeoutCmd, rTimer := _timerCmd);
          // inc step counter
         _stepCmd := _stepCmd + 1;
        ELSE
          // check error ?
          IF (_readRobotData.Error)
          THEN
            ErrorID     := _readRobotData.ErrorID;
            ErrorAddTxt := _readRobotData.ErrorAddTxt;;
          END_IF
          // timeout exceeded ?
          IF (CheckTimeout(_timerCmd) = RobotLibraryConstants.OK)
          THEN
            ErrorID     := RobotLibraryErrorIdEnum.ERR_TIMEOUT_CMD;
            ErrorAddTxt := CONCAT('_stepCmd = ' , DINT_TO_STRING(_stepCmd));
          END_IF
        END_IF

    07: IF (( NOT _readRobotData.Busy  ) AND
            (     _readRobotData.Done  ))
        THEN
          // Reset busy flag
          Busy := FALSE;
          // set initialized flag
          Initialized := TRUE;
          // start function block
         _readRobotData.Execute := FALSE;
          // set timeout
          SetTimeout(PT := _timeoutCmd, rTimer := _timerCmd);
          // inc step counter
         _stepCmd := _stepCmd + 1;
         ELSE
           // check error ?
           IF (_readRobotData.Error)
           THEN
             ErrorID     := _readRobotData.ErrorID;
             ErrorAddTxt := _readRobotData.ErrorAddTxt;;
           END_IF

           // timeout exceeded ?
           IF (CheckTimeout(_timerCmd) = RobotLibraryConstants.OK)
           THEN
             ErrorID     := RobotLibraryErrorIdEnum.ERR_TIMEOUT_CMD;
             ErrorAddTxt := CONCAT('_stepCmd = ' , DINT_TO_STRING(_stepCmd));
           END_IF
         END_IF

    08:  // Update Initialized state
         Initialized := NOT Synchronized;

         // Wait for task disable
         IF ( NOT Enable)
         THEN
           // Reset active command register
           AxesGroup.Acyclic.ActiveCommandRegister.Reset();
           // reset internal variables
           Reset(AxesGroup := AxesGroup);
           // Reset step counter
          _stepCmd := 0;
           // finished okay
           OnExecRun := RobotLibraryConstants.OK;
         END_IF

  ELSE
    // invalid step
    ErrorID     := RobotLibraryErrorIdEnum.ERR_INVALID_STEP;
    ErrorAddTxt := CONCAT('_stepCmd = ' , DINT_TO_STRING(_stepCmd));
  END_CASE

END_METHOD

METHOD PRIVATE ParseRecvPayload
VAR_IN_OUT
  /// Robot assignment of function
  AxesGroup    : AxesGroup;
  /// Inputs of PLC for communication from RC
  RobotInData  : ARRAY[0..RobotLibraryParameter.ROBOT_IN_DATA_MAX ] OF BYTE;
END_VAR

VAR
  /// internal index
 _idx             : DINT;
  /// temporary DWORD
 _tmpDword        : DWORD;
  /// length of data block
 _dataBlockLength : UINT;
  /// internal payload length
 _payLoadLen      : DWORD;
  /// internal payload pointer
 _payLoadPtr      : DWORD;
  /// sequence counter
 _seqCount        : DINT;
END_VAR

  // Reset payload
  RecvData.Reset();
  // Copy inputs to payload
  SysDepMemCpy( pDest := ADR(RecvData.Payload) , pSrc  := ADR(RobotInData), DataLen := RobotLibraryParameter.ROBOT_IN_DATA_MAX +1);

  // check new data to receive ?
  IF ( Telegram.RobToPlc.Sequence[0].Header.SEQ_ACK <> AxesGroup.State.LastACK[0]) {warning 'ToDo: handle 2nd sequence'}
  THEN
    // delete old telegram data
    SysDepMemSet(pDest := ADR(Telegram.RobToPlc), Value := 0 , DataLen := SIZEOF(Telegram.RobToPlc));
  END_IF

  ParseRecvPayloadHeader        ( AxesGroup := AxesGroup);
  ParseRecvPayloadCyclic        ( AxesGroup := AxesGroup);
  ParseRecvPayloadCyclicOptional( AxesGroup := AxesGroup);
  ParseRecvPayloadSequence      ( AxesGroup := AxesGroup);
  ParseRecvPayloadFooter        ( AxesGroup := AxesGroup);
  ParseRecvPayloadLogging       ( AxesGroup := AxesGroup);

  AxesGroup.State.LastACK[0] := Telegram.RobToPlc.Sequence[0].Header.SEQ_ACK;
  AxesGroup.State.LastACK[1] := Telegram.RobToPlc.Sequence[1].Header.SEQ_ACK;

END_METHOD

METHOD PRIVATE ParseRecvPayloadCyclic
VAR_IN_OUT
  /// Robot assignment of function
  AxesGroup: AxesGroup;
END_VAR

END_METHOD

METHOD PRIVATE ParseRecvPayloadCyclicOptional
VAR_IN_OUT
  /// Robot assignment of function
  AxesGroup    : AxesGroup;
END_VAR

VAR
  /// internal index for loops
 _idx : DINT;
END_VAR

  // AxesGroup.OptionalCyclic.RobToPlc.SubProgramData {{{
  IF ( AxesGroup.CyclicOptional.RobToPlc.SubProgramData.Active )
  THEN
    FOR _idx := 0 TO 25 {warning 'Add contant for DataMax'}
    DO
      Telegram.RobToPlc.CyclicOptional.SubProgramData.Data[_idx] := RecvData.GetByte();
    END_FOR
  END_IF
  // }}}

  // AxesGroup.OptionalCyclic.RobToPlc.CartesianPos {{{
  IF ( AxesGroup.CyclicOptional.RobToPlc.CartesianPosition.Active )
  THEN
    Telegram.RobToPlc.CyclicOptional.CartesianPosition.X                    := RecvData.GetReal();
    Telegram.RobToPlc.CyclicOptional.CartesianPosition.Y                    := RecvData.GetReal();
    Telegram.RobToPlc.CyclicOptional.CartesianPosition.Z                    := RecvData.GetReal();
    Telegram.RobToPlc.CyclicOptional.CartesianPosition.Rx                   := RecvData.GetReal();
    Telegram.RobToPlc.CyclicOptional.CartesianPosition.Ry                   := RecvData.GetReal();
    Telegram.RobToPlc.CyclicOptional.CartesianPosition.Rz                   := RecvData.GetReal();
    Telegram.RobToPlc.CyclicOptional.CartesianPosition.Config               := RecvData.GetWord();
    Telegram.RobToPlc.CyclicOptional.CartesianPosition.Turns_J2_J1          := RecvData.GetByte();
    Telegram.RobToPlc.CyclicOptional.CartesianPosition.Turns_J4_J3          := RecvData.GetByte();
    Telegram.RobToPlc.CyclicOptional.CartesianPosition.Turns_J6_J5          := RecvData.GetByte();
    Telegram.RobToPlc.CyclicOptional.CartesianPosition.Turns_E1             := RecvData.GetByte();
    Telegram.RobToPlc.CyclicOptional.CartesianPosition.E1                   := RecvData.GetReal();
    Telegram.RobToPlc.CyclicOptional.CartesianPosition.ToolNo               := RecvData.GetUsint();
    Telegram.RobToPlc.CyclicOptional.CartesianPosition.FrameNo              := RecvData.GetUsint();
    Telegram.RobToPlc.CyclicOptional.CartesianPosition.CurrentlyUsedToolNo  := RecvData.GetUsint();
    Telegram.RobToPlc.CyclicOptional.CartesianPosition.CurrentlyUsedFrameNo := RecvData.GetUsint();
    Telegram.RobToPlc.CyclicOptional.CartesianPosition.Reserve_1            := RecvData.GetByte();
    Telegram.RobToPlc.CyclicOptional.CartesianPosition.Reserve_2            := RecvData.GetByte();
  END_IF
  // }}}

  // AxesGroup.OptionalCyclic.RobToPlc.JointPosition {{{
  IF ( AxesGroup.CyclicOptional.RobToPlc.JointPosition.Active )
  THEN
    Telegram.RobToPlc.CyclicOptional.JointPosition.J1         := RecvData.GetReal();
    Telegram.RobToPlc.CyclicOptional.JointPosition.J2         := RecvData.GetReal();
    Telegram.RobToPlc.CyclicOptional.JointPosition.J3         := RecvData.GetReal();
    Telegram.RobToPlc.CyclicOptional.JointPosition.J4         := RecvData.GetReal();
    Telegram.RobToPlc.CyclicOptional.JointPosition.J5         := RecvData.GetReal();
    Telegram.RobToPlc.CyclicOptional.JointPosition.J6         := RecvData.GetReal();
    Telegram.RobToPlc.CyclicOptional.JointPosition.E1         := RecvData.GetReal();
    Telegram.RobToPlc.CyclicOptional.JointPosition.E1_Reserve := RecvData.GetWord();
  END_IF
  // }}}

  // AxesGroup.OptionalCyclic.RobToPlc.CartesianForce {{{
  IF ( AxesGroup.CyclicOptional.RobToPlc.Force.Active )
  THEN
    Telegram.RobToPlc.CyclicOptional.Force.X  := RecvData.GetReal();
    Telegram.RobToPlc.CyclicOptional.Force.Y  := RecvData.GetReal();
    Telegram.RobToPlc.CyclicOptional.Force.Z  := RecvData.GetReal();
    Telegram.RobToPlc.CyclicOptional.Force.Rx := RecvData.GetReal();
    Telegram.RobToPlc.CyclicOptional.Force.Ry := RecvData.GetReal();
    Telegram.RobToPlc.CyclicOptional.Force.Rz := RecvData.GetReal();
  END_IF
  // }}}

  // AxesGroup.OptionalCyclic.RobToPlc.Current {{{
  IF ( AxesGroup.CyclicOptional.RobToPlc.Current.Active )
  THEN
    Telegram.RobToPlc.CyclicOptional.Current.J1  := RecvData.GetReal();
    Telegram.RobToPlc.CyclicOptional.Current.J2  := RecvData.GetReal();
    Telegram.RobToPlc.CyclicOptional.Current.J3  := RecvData.GetReal();
    Telegram.RobToPlc.CyclicOptional.Current.J4  := RecvData.GetReal();
    Telegram.RobToPlc.CyclicOptional.Current.J5  := RecvData.GetReal();
    Telegram.RobToPlc.CyclicOptional.Current.J6  := RecvData.GetReal();
  END_IF

  // AxesGroup.OptionalCyclic.RobToPlc.CartesianPosExt {{{
  IF ( AxesGroup.CyclicOptional.RobToPlc.CartesianPositionExt.Active )
  THEN
    Telegram.RobToPlc.CyclicOptional.CartesianPositionExt.E2 := RecvData.GetReal();
    Telegram.RobToPlc.CyclicOptional.CartesianPositionExt.E3 := RecvData.GetReal();
    Telegram.RobToPlc.CyclicOptional.CartesianPositionExt.E4 := RecvData.GetReal();
    Telegram.RobToPlc.CyclicOptional.CartesianPositionExt.E5 := RecvData.GetReal();
    Telegram.RobToPlc.CyclicOptional.CartesianPositionExt.E6 := RecvData.GetReal();
  END_IF
  // }}}

  // AxesGroup.OptionalCyclic.RobToPlc.JointPosition {{{
  IF ( AxesGroup.CyclicOptional.RobToPlc.JointPositionExt.Active )
  THEN
    Telegram.RobToPlc.CyclicOptional.JointPositionExt.E2 := RecvData.GetReal();
    Telegram.RobToPlc.CyclicOptional.JointPositionExt.E3 := RecvData.GetReal();
    Telegram.RobToPlc.CyclicOptional.JointPositionExt.E4 := RecvData.GetReal();
    Telegram.RobToPlc.CyclicOptional.JointPositionExt.E5 := RecvData.GetReal();
    Telegram.RobToPlc.CyclicOptional.JointPositionExt.E6 := RecvData.GetReal();
  END_IF
  // }}}

  // AxesGroup.OptionalCyclic.RobToPlc.CartesianForceExt {{{
  IF ( AxesGroup.CyclicOptional.RobToPlc.ForceExt.Active )
  THEN
    Telegram.RobToPlc.CyclicOptional.ForceExt.E1  := RecvData.GetReal();
    Telegram.RobToPlc.CyclicOptional.ForceExt.E2  := RecvData.GetReal();
    Telegram.RobToPlc.CyclicOptional.ForceExt.E3  := RecvData.GetReal();
    Telegram.RobToPlc.CyclicOptional.ForceExt.E4  := RecvData.GetReal();
    Telegram.RobToPlc.CyclicOptional.ForceExt.E5  := RecvData.GetReal();
    Telegram.RobToPlc.CyclicOptional.ForceExt.E6  := RecvData.GetReal();
  END_IF
  // }}}

  // AxesGroup.OptionalCyclic.RobToPlc.CurrentExt {{{
  IF ( AxesGroup.CyclicOptional.RobToPlc.CurrentExt.Active )
  THEN
    Telegram.RobToPlc.CyclicOptional.CurrentExt.E1  := RecvData.GetReal();
    Telegram.RobToPlc.CyclicOptional.CurrentExt.E2  := RecvData.GetReal();
    Telegram.RobToPlc.CyclicOptional.CurrentExt.E3  := RecvData.GetReal();
    Telegram.RobToPlc.CyclicOptional.CurrentExt.E4  := RecvData.GetReal();
    Telegram.RobToPlc.CyclicOptional.CurrentExt.E5  := RecvData.GetReal();
    Telegram.RobToPlc.CyclicOptional.CurrentExt.E6  := RecvData.GetReal();
  END_IF
  // }}}

END_METHOD

METHOD PRIVATE ParseRecvPayloadFooter
VAR_IN_OUT
  /// Robot assignment of function
  AxesGroup : AxesGroup;
END_VAR

VAR
  /// index of lifesign in footer
  _lifeSignIdxFooter : DINT;
END_VAR

  IF (( _parCfg.Com.TelegramLengthRobToPlc >= 1                                           ) AND
      ( _parCfg.Com.TelegramLengthRobToPlc <= RobotLibraryParameter.ROBOT_IN_DATA_MAX + 1 ))
  THEN
    // set index of last byte
   _lifeSignIdxFooter := _parCfg.Com.TelegramLengthRobToPlc -1;

    Telegram.RobToPlc.Footer.LifeSign := GetHalfeByteHi(RecvData.Payload[_lifeSignIdxFooter]);
  END_IF

END_METHOD

METHOD PRIVATE ParseRecvPayloadHeader
VAR_IN_OUT
  /// Robot assignment of function
  AxesGroup    : AxesGroup;
END_VAR

  // Version
  Telegram.RobToPlc.Header.SRCIVersion := ByteToVersion(RecvData.GetByte());
  // Connection alive signal
  Telegram.RobToPlc.Header.LifeSign    := RecvData.GetHalfeByte2(IncPayloadPtr := TRUE);
  // Reserved byte
  Telegram.RobToPlc.Header.Reserved       := RecvData.GetByte();
  // Initialization and Telegram control state
  Telegram.RobToPlc.Header.TelegramState  := RecvData.GetUsint();
  // Combination of various RA related states.
  Telegram.RobToPlc.Header.StatusRobotArm := RecvData.GetDword();
  // Actual override in percentage encoding
  Telegram.RobToPlc.Header.Override       := RecvData.GetUint();

END_METHOD

METHOD PRIVATE ParseRecvPayloadLogging
VAR_IN_OUT
  /// Robot assignment of function
  AxesGroup    : AxesGroup;
END_VAR

VAR
  /// internal sequence index for loops
  _seqIdx : DINT;
  /// internal fragment index for loops
  _fragIdx : DINT;
END_VAR
